		//Wait for Delay, copy Data and then next step
		IF NOT fbMBRead_FC4.bBusy AND NOT fbMBRead_FC4.bError AND timDelay.Q THEN
			//Connecotor State
			arrConnectorState[wConnectorInProgress] := arrBuffer_FC4[1];
			//Connector Power
			fbConvertWordToDord(wInputValue_1:= arrBuffer_FC4[5], wInputValue_2:= arrBuffer_FC4[6], eByteOrderForConvert:= eByteOrder.eBigEndian, dwOutputValue=> );
				arrPowerConnector[wConnectorInProgress] := fbConvertWordToDord.dwOutputValue;
			//Charging Time in Seconds
			arrChargingTime[wConnectorInProgress] := arrBuffer_FC4[7];
			//Energy Session
			arrEnergySession[wConnectorInProgress] := WORD_TO_REAL(arrBuffer_FC4[8]) / 100;
			//SOC from the Car
			arrSOCCar[wConnectorInProgress] := arrBuffer_FC4[9] / 100;
			//Go to Next Step
			fbMBRead_FC4.bExecute := FALSE;
				timDelay.IN := FALSE;		
					iStateModbusRead := 3;
		END_IF	

		//Error or Timeout
		IF FPError_FC_4.Q OR timTimeout.Q THEN
			iStateModbusError := 300;
		END_IF
		
	3://Wait 1 Step to reset the delay counter befor start to write
		iStateModbus_CP := iStateModbusRead;
		
			iStateModbusWrite := 1;
				//-1 because 0 is the Init Step for Read
				iStateModbusRead := - 1;
				
			//Error on Master, changes on Inputs or Timeout
		 	IF timTimeout.Q THEN 
				iStateModbusError := 300; 
					 
			END_IF
	
END_CASE

(*------------------------------------------------------------------Error and Warning----------------------------------------------------------------------------*)	
 
IF wStationState = 10 OR arrConnectorState[1] = 10 OR arrConnectorState[2] = 10 OR arrConnectorState[3] = 10 OR arrConnectorState[4] = 10 THEN bErrorCS := TRUE; ELSE bErrorCS := FALSE; END_IF  

IF timDissableFunctions.Q THEN fbCS.bWarning := TRUE; fbCS.iWarningCode := 0; ELSE fbCS.bWarning := FALSE; END_IF   
	IF Lynus_Standards.GVL_Energy.stNumberOfDevices.diNumberOfECS > Constants_Energy.diMaxNumberOfElectricChargingStations OR bErrorCS OR bMBTCPError THEN 
		fbCS.bError := TRUE;
	ELSE 
		fbCS.bError := FALSE;
			fbCS.iErrorCode := 0;
	END_IF

IF Lynus_Standards.GVL_Energy.stNumberOfDevices.diNumberOfECS > Constants_Energy.diMaxNumberOfElectricChargingStations THEN fbCS.iErrorCode := 1;
ELSIF bErrorCS OR bMBTCPError THEN fbCS.iErrorCode := 0; END_IF

(*------------------------------------------------------------------Logic----------------------------------------------------------------------------*)

//Calcualte the total SOC if we have more then 1 battery in our system
diNumberOfActiveBatterys := 0;
	dwSumSOC := 0;
		FOR liLPBatteryData := 1 TO Constants_Energy.diMaxNumberOfBatterys BY 1 DO
			IF Lynus_Standards.GVL_Energy.stDataOfBatterys[diNrOfEMS_IN,liLPBatteryData].bEnabled THEN diNumberOfActiveBatterys := diNumberOfActiveBatterys + 1; END_IF
				dwSumSOC := dwSumSOC + Lynus_Standards.GVL_Energy.stDataOfBatterys[diNrOfEMS_IN,liLPBatteryData].dwSOC;
		END_FOR
	
IF diNumberOfActiveBatterys > 0 THEN
	fbCS.dwBatterySOC := DINT_TO_DWORD(DWORD_TO_DINT(dwSumSOC) / diNumberOfActiveBatterys);
ELSE
	fbCS.dwBatterySOC := 100;	//When we have no battery in the ems system
END_IF

//Check if one or more Batterysystems or batteryinverter make island mode
diNumberOfBatteryInverterInEPO := 0;
	FOR liLPInEPO := 1 TO Constants_Energy.diMaxNumberOfBatteryInverters BY 1 DO
		IF Lynus_Standards.GVL_Energy.stDataOfBatteryInverters[diNrOfEMS_IN,liLPInEPO].bWorkOnIslandMode THEN fbCS.bEPOIsActive := TRUE; diNumberOfBatteryInverterInEPO := diNumberOfBatteryInverterInEPO + 1; END_IF
	END_FOR 
		IF diNumberOfBatteryInverterInEPO <= 0 THEN fbCS.bEPOIsActive := FALSE; END_IF

//Digital input for external lock signal
fbDIExternalLock(bInvers:= FALSE, bSignal=> );

//Car connected to the ECS  
IF arrConnectorState[1] = 2 OR arrConnectorState[2] = 2 OR arrConnectorState[3] = 2 OR arrConnectorState[4] = 2 OR
	 arrConnectorState[1] = 3 OR arrConnectorState[2] = 3 OR arrConnectorState[3] = 3 OR arrConnectorState[4] = 3 OR 
		arrConnectorState[1] = 6 OR arrConnectorState[2] = 6 OR arrConnectorState[3] = 6 OR arrConnectorState[4] = 6 THEN 
		fbCS.bCarConnected := TRUE; 
ELSE 
		fbCS.bCarConnected := FALSE; 
END_IF 

//Charging time and SOC from the Car
fbCS.arrSocketChargingTimeInput[1] :=  arrChargingTime[1] / 60;
fbCS.arrSocketChargingTimeInput[2] :=  arrChargingTime[2] / 60;
fbCS.arrSocketChargingTimeInput[3] :=  arrChargingTime[3] / 60;
fbCS.arrSocketChargingTimeInput[4] :=  arrChargingTime[4] / 60;

fbCS.arrSOCCar[1] := arrSOCCar[1];
fbCS.arrSOCCar[2] := arrSOCCar[2];
fbCS.arrSOCCar[3] := arrSOCCar[3];
fbCS.arrSOCCar[4] := arrSOCCar[4];

//Mode 3 State
fbCS.arrSocketMode3StateECS[1] := '';
fbCS.arrSocketMode3StateECS[2] := '';
fbCS.arrSocketMode3StateECS[3] := '';
fbCS.arrSocketMode3StateECS[4] := '';
//ECS is Free
IF arrConnectorState[1] = 0 THEN fbCS.arrSocketMode3StateECS[1] := 'A'; END_IF
IF arrConnectorState[2] = 0 THEN fbCS.arrSocketMode3StateECS[2] := 'A'; END_IF
IF arrConnectorState[3] = 0 THEN fbCS.arrSocketMode3StateECS[3] := 'A'; END_IF
IF arrConnectorState[4] = 0 THEN fbCS.arrSocketMode3StateECS[4] := 'A'; END_IF
//ECS Car Connected
IF arrConnectorState[1] = 2 OR arrConnectorState[1] = 6 THEN fbCS.arrSocketMode3StateECS[1] := 'B1'; END_IF
IF arrConnectorState[2] = 2 OR arrConnectorState[2] = 6 THEN fbCS.arrSocketMode3StateECS[2] := 'B1'; END_IF
IF arrConnectorState[3] = 2 OR arrConnectorState[3] = 6 THEN fbCS.arrSocketMode3StateECS[3] := 'B1'; END_IF
IF arrConnectorState[4] = 2 OR arrConnectorState[4] = 6 THEN fbCS.arrSocketMode3StateECS[4] := 'B1'; END_IF
//ECS Car is Charging
IF arrConnectorState[1] = 3 THEN fbCS.arrSocketMode3StateECS[1] := 'C2'; END_IF
IF arrConnectorState[2] = 3 THEN fbCS.arrSocketMode3StateECS[2] := 'C2'; END_IF
IF arrConnectorState[3] = 3 THEN fbCS.arrSocketMode3StateECS[3] := 'C2'; END_IF
IF arrConnectorState[4] = 3 THEN fbCS.arrSocketMode3StateECS[4] := 'C2'; END_IF

//Functionblock ECS
fbCS(
	bEnable:= bEnable AND NOT timDissableFunctions.Q, 
	bError:= ,
	bWarning := ,
	bEPOIsActive:= , 
	bExternalLock:= fbDIExternalLock.bSignal, 
	bCarConnected:= , 
	bWriteWithDelay:= TRUE, 
	bCalculateEnergySession:= ,
	iErrorCode:= , 
	iWarningCode:= , 
	arrSocketChargingTimeInput:= ,
	arrSOCCar:= , 
	dwBatterySOC:= , 
	lrTotalCounterEnergy_Consumption:= , 
	lrTotalCounterEnergy_Production:= , 
	lrCounterEnergyT1_Consumption:= , 
	lrCounterEnergyT2_Consumption:= , 
	lrCounterEnergyT1_Production:= , 
	lrCounterEnergyT2_Production:= , 
	lrTotalPowerECS:= , 
	arrSocketEnergySession:= ,
	rTargetPower:= Lynus_Standards.GVL_Energy.stDataElectricChargingStations[diNrOfEMS_IN,diNrOfECS_OUT].rTargetPowerEMS, 
	rSupplyVoltage:= 692, 
	rMinCurrent:= 7.5, 
	tTimDelayOutput:= T#5S, 
	tDelayError:= T#5S,
	arrSocketMode3StateECS:= ,
	arrSocketPowerECS:= ,
	stSetupECS:= stSetupECS, 
	stDataECSOut=> , 
	stDataECSOutDelay=> stDataECS);

dwTargetPower := REAL_TO_DWORD((stSetupECS.rMaxPower * fbCS.stDataECSOut.rTargetPower) / 100);
	dwTargetPower := dwTargetPower * 1000;

//Real time Power for Output
lrTotalPowerECSRealTime := fbCS.stDataECSOut.lrTotalPower;
	
(*------------------------------------------------------------------------------------------State Machine Write---------------------------------------------------------------------------------------------*)	

CASE iStateModbusWrite OF	

	1://Set the charging power (Reg 0)
		iStateModbus_CP := iStateModbusWrite;
		
			fbMBWrite_FC16.nQuantity := 2;
				fbMBWrite_FC16.nMBAddr := 0;
					fbMBWrite_FC16.bExecute := TRUE;
						fbMBWrite_FC16.nUnitID := byUnitID;
		
		//Prepear the sending Data. Charging Power for the charging station. 
		//Charging power
		fbConvertDwordToWord(dwInputValue:= dwTargetPower, eByteOrderForConvert:= eByteOrder.eBigEndian, wOutputValue_1=> arrBuffer_FC16[1], wOutputValue_2=> arrBuffer_FC16[2]);
		
		IF fbMBWrite_FC16.bBusy THEN timDelay.IN := TRUE; END_IF

		//Wait for Delay and then next step
		IF NOT fbMBWrite_FC16.bBusy AND NOT fbMBWrite_FC16.bError AND timDelay.Q THEN
			fbMBWrite_FC16.bExecute := FALSE;
				timDelay.IN := FALSE;
					bMBTCPError := FALSE; 
						//Restart from new with the Read out part
						iStateModbusRead := 1;
							iStateModbusWrite := 0;
								wConnectorInProgress := wConnectorInProgress + 1;
									IF wConnectorInProgress > 4 OR wConnectorInProgress > wNumberOfConnectors THEN wConnectorInProgress := 1; END_IF
		END_IF
				
		//Error or Timout
		IF FPError_FC_16.Q OR timTimeout.Q THEN
			iStateModbusError := 300;
		END_IF
		
END_CASE	
	
(*------------------------------------------------------------------------------------------State Machine Error---------------------------------------------------------------------------------------------*)	

CASE iStateModbusError OF
	
	300://Error
		iStateModbus_CP := iStateModbusError;
			timDelay.IN := FALSE;
				fbMBRead_FC4.bExecute := FALSE;
					fbMBWrite_FC16.bExecute := FALSE;
						bMBTCPError := TRUE; 		
							//Restart from new with the Read out part after an Error
							iStateModbusRead := 1;	
								iStateModbusError := 0;
									iStateModbusWrite := 0;
						
END_CASE

(*------------------------------------------------------------------------------------------Modbus TCP Functions---------------------------------------------------------------------------------------------*)

fbMBRead_FC4(sIPAddr:= sIPAdress, nTCPPort:= 502,cbLength:= SIZEOF(arrBuffer_FC4), pDestAddr:= ADR(arrBuffer_FC4), tTimeout:= T#10S );
	FPError_FC_4(CLK:= fbMBRead_FC4.bError, Q=> );		

fbMBWrite_FC16(sIPAddr:= sIPAdress, nTCPPort:= 502, cbLength:= SIZEOF(arrBuffer_FC16), pSrcAddr:= ADR(arrBuffer_FC16), tTimeout:= T#10S);	
	FPError_FC_16(CLK:= fbMBWrite_FC16.bError, Q=> );

(*-----------------------------------------------------------Handle data to Global structure for electric charging stations-----------------------------------------------------------------*)

//Delte al old Data on GVL after a online change or change on the variable diNrOfEMS_IDOD
IF diNrOfEMS_IN <> diNrOfEMS_IN_CP AND iStateGVLData = 0 THEN iStateGVLData := 10; END_IF 

CASE iStateGVLData OF
	
	0://Init Step
		byWaitInStep := 0;
			diCounterForGVL := 1;
	
	1://Wait for 4 Steps before clean al Data on GVL
		byWaitInStep := byWaitInStep + 1;
			IF byWaitInStep >= 4 AND fbNumberDevice.bNumberIsCalculatet THEN iStateGVLData := 2; END_IF
				//To much Devices, back to the Init step
				IF byWaitInStep >= 4 AND NOT fbNumberDevice.bNumberIsCalculatet THEN iStateGVLData := 0; END_IF	
			
	2://Clear all Data in GVL
		FOR diLPForGVL := 1 TO Constants_Energy.diMaxNumberOfEMS BY 1 DO 
			Lynus_Standards.GVL_Energy.stDataElectricChargingStations[diLPForGVL,diCounterForGVL].bEnabled := FALSE;
				Lynus_Standards.GVL_Energy.stDataElectricChargingStations[diLPForGVL,diCounterForGVL].bIsControllable := FALSE;
					Lynus_Standards.GVL_Energy.stDataElectricChargingStations[diLPForGVL,diCounterForGVL].byErrorWarning := 0;
						Lynus_Standards.GVL_Energy.stDataElectricChargingStations[diLPForGVL,diCounterForGVL].byPriority := 0;
							Lynus_Standards.GVL_Energy.stDataElectricChargingStations[diLPForGVL,diCounterForGVL].lrPower := 0;
								Lynus_Standards.GVL_Energy.stDataElectricChargingStations[diLPForGVL,diCounterForGVL].lrPowerConsumption := 0;
									Lynus_Standards.GVL_Energy.stDataElectricChargingStations[diLPForGVL,diCounterForGVL].lrPowerProduction := 0;
										Lynus_Standards.GVL_Energy.stDataElectricChargingStations[diLPForGVL,diCounterForGVL].rMaxPower := 0;
											//Set also the target value from ems back here to 0 and not in EMS function because EMS is in Standy when we have a online change (Problem when we delete a ems function and make a online change)
											Lynus_Standards.GVL_Energy.stDataElectricChargingStations[diLPForGVL,diCounterForGVL].rTargetPowerEMS := 0;	
		END_FOR
		
			//Counter for ECS
			diCounterForGVL := diCounterForGVL + 1;
				diCounterForGVL := LIMIT(0,diCounterForGVL,Constants_Energy.diMaxNumberOfElectricChargingStations);
					//Back to the init step
					IF diCounterForGVL >= Constants_Energy.diMaxNumberOfElectricChargingStations THEN iStateGVLData := 0; END_IF

	10://Clear old Data on GVL 		
		Lynus_Standards.GVL_Energy.stDataElectricChargingStations[diNrOfEMS_IN_CP,diNrOfECS_OUT].bEnabled := FALSE;
			Lynus_Standards.GVL_Energy.stDataElectricChargingStations[diNrOfEMS_IN_CP,diNrOfECS_OUT].bIsControllable := FALSE;
				Lynus_Standards.GVL_Energy.stDataElectricChargingStations[diNrOfEMS_IN_CP,diNrOfECS_OUT].byErrorWarning := 0;
					Lynus_Standards.GVL_Energy.stDataElectricChargingStations[diNrOfEMS_IN_CP,diNrOfECS_OUT].byPriority := 0;
						Lynus_Standards.GVL_Energy.stDataElectricChargingStations[diNrOfEMS_IN_CP,diNrOfECS_OUT].lrPower := 0;
							Lynus_Standards.GVL_Energy.stDataElectricChargingStations[diNrOfEMS_IN_CP,diNrOfECS_OUT].lrPowerConsumption := 0;
								Lynus_Standards.GVL_Energy.stDataElectricChargingStations[diNrOfEMS_IN_CP,diNrOfECS_OUT].lrPowerProduction := 0;
									Lynus_Standards.GVL_Energy.stDataElectricChargingStations[diNrOfEMS_IN_CP,diNrOfECS_OUT].rMaxPower := 0;
									
		diNrOfEMS_IN_CP := diNrOfEMS_IN;
			//Back to the init step
			iStateGVLData := 0;

END_CASE 	 

IF diNrOfECS_OUT > 0 AND fbNumberDevice.bNumberIsCalculatet AND diNrOfEMS_IN > 0 THEN
	Lynus_Standards.GVL_Energy.stDataElectricChargingStations[diNrOfEMS_IN,diNrOfECS_OUT].bEnabled := fbCS.stDataECSOut.bEnabled;
		Lynus_Standards.GVL_Energy.stDataElectricChargingStations[diNrOfEMS_IN,diNrOfECS_OUT].bIsControllable := TRUE;
			Lynus_Standards.GVL_Energy.stDataElectricChargingStations[diNrOfEMS_IN,diNrOfECS_OUT].byErrorWarning := fbCS.stDataECSOut.byErrorWarning;
				Lynus_Standards.GVL_Energy.stDataElectricChargingStations[diNrOfEMS_IN,diNrOfECS_OUT].byPriority := fbCS.stDataECSOut.byPriority;
					Lynus_Standards.GVL_Energy.stDataElectricChargingStations[diNrOfEMS_IN,diNrOfECS_OUT].lrPower := fbCS.stDataECSOut.lrTotalPower;
						Lynus_Standards.GVL_Energy.stDataElectricChargingStations[diNrOfEMS_IN,diNrOfECS_OUT].lrPowerConsumption := fbCS.stDataECSOut.lrTotalPowerConsumption;
							Lynus_Standards.GVL_Energy.stDataElectricChargingStations[diNrOfEMS_IN,diNrOfECS_OUT].lrPowerProduction := fbCS.stDataECSOut.lrTotalPowerProduction;
								Lynus_Standards.GVL_Energy.stDataElectricChargingStations[diNrOfEMS_IN,diNrOfECS_OUT].rMaxPower := fbCS.stDataECSOut.rMaxPower;	
END_IF 

(*----------------------------------------------------------Save persistent data----------------------------------------------------------------*)

arrPD[1](lrValue:= BOOL_TO_LREAL(bEnable), bEventBasedActive=> );
arrPD[2](lrValue:= BOOL_TO_LREAL(bPowerDataInvers), bEventBasedActive=> );
arrPD[3](lrValue:= DINT_TO_LREAL(diNrOfEMS_IN), bEventBasedActive=> );
arrPD[4](lrValue:= DINT_TO_LREAL(diNrOfEM_IN_CS), bEventBasedActive=> );
arrPD[5](lrValue:= BOOL_TO_LREAL(stSetupECS.bManualyOn), bEventBasedActive=> );
arrPD[6](lrValue:= BOOL_TO_LREAL(stSetupECS.bOnEmergPowerOff), bEventBasedActive=> );
arrPD[7](lrValue:= BYTE_TO_LREAL(stSetupECS.byCSMinPower), bEventBasedActive=> );
arrPD[8](lrValue:= BYTE_TO_LREAL(stSetupECS.byDisableSOC), bEventBasedActive=> );
arrPD[9](lrValue:= BYTE_TO_LREAL(stSetupECS.byEnableSOC), bEventBasedActive=> );
arrPD[10](lrValue:= BYTE_TO_LREAL(stSetupECS.byManualyTargetPower), bEventBasedActive=> );
arrPD[11](lrValue:= BYTE_TO_LREAL(stSetupECS.byPriority), bEventBasedActive=> );
arrPD[12](lrValue:= REAL_TO_LREAL(stSetupECS.rMaxPower), bEventBasedActive=> );
arrPD[13](lrValue:= DINT_TO_LREAL(diNrOfEMS_IN_CP), bEventBasedActive=> );
arrPD[14](lrValue:= BYTE_TO_LREAL(byUnitID), bEventBasedActive=> );
fbPDString(sText:= sIPAdress, bEventBasedActive=> );

END_FUNCTION_BLOCK

// ---- POUs/prgCS2.TcPOU
PROGRAM prgCS2
VAR
	fbAlfen1					: FB_ECS_Alfen_NG9xx_Platform;						//{#lynus.ag#()}
	fbAlfen2					: FB_ECS_Alfen_NG9xx_Platform;						//{#lynus.ag#()}
	fbAlfen3					: FB_ECS_Alfen_NG9xx_Platform;						//{#lynus.ag#()}
	fbAlfen4					: FB_ECS_Alfen_NG9xx_Platform;						//{#lynus.ag#()}
	fbAlfen5					: FB_ECS_Alfen_NG9xx_Platform;						//{#lynus.ag#()}
	fbAlfen6					: FB_ECS_Alfen_NG9xx_Platform;						//{#lynus.ag#()}
	fbAlfen7					: FB_ECS_Alfen_NG9xx_Platform;						//{#lynus.ag#()}
	fbAlfen8					: FB_ECS_Alfen_NG9xx_Platform;						//{#lynus.ag#()}
	fbAlfen9					: FB_ECS_Alfen_NG9xx_Platform;						//{#lynus.ag#()}
	fbAlfen10					: FB_ECS_Alfen_NG9xx_Platform;						//{#lynus.ag#()}
	
	bSManualyOn_UV1_1			: BOOL;												//{#lynus.ag#()}
	bySManualyTargetPowerUV1_1	: BYTE;												//{#lynus.ag#()}
	byErrorWarningUV1_1			: BYTE;												//{#lynus.ag#()}
	rChargingTimeInMinUV1_1		: REAL;												//{#lynus.ag#()}
	lrPowerUV1_1				: LREAL;											//{#lynus.ag#()}
	wStateUV1_1					: WORD;												//{#lynus.ag#()}
	lrEnergySessionUV1_1		: LREAL;											//{#lynus.ag#()}
	lrTotalEnergyUV1_1			: LREAL;											//{#lynus.ag#()}
	
	bSManualyOn_UV1_2			: BOOL;												//{#lynus.ag#()}
	bySManualyTargetPowerUV1_2	: BYTE;												//{#lynus.ag#()}
	byErrorWarningUV1_2			: BYTE;												//{#lynus.ag#()}
	rChargingTimeInMinUV1_2		: REAL;												//{#lynus.ag#()}
	lrPowerUV1_2				: LREAL;											//{#lynus.ag#()}
	wStateUV1_2					: WORD;												//{#lynus.ag#()}
	lrEnergySessionUV1_2		: LREAL;											//{#lynus.ag#()}
	lrTotalEnergyUV1_2			: LREAL;											//{#lynus.ag#()}
	
	bSManualyOn_UV1_3			: BOOL;												//{#lynus.ag#()}
	bySManualyTargetPowerUV1_3	: BYTE;												//{#lynus.ag#()}
	byErrorWarningUV1_3			: BYTE;												//{#lynus.ag#()}
	rChargingTimeInMinUV1_3		: REAL;												//{#lynus.ag#()}
	lrPowerUV1_3				: LREAL;											//{#lynus.ag#()}
	wStateUV1_3					: WORD;												//{#lynus.ag#()}
	lrEnergySessionUV1_3		: LREAL;											//{#lynus.ag#()}
	lrTotalEnergyUV1_3			: LREAL;											//{#lynus.ag#()}
	
	bSManualyOn_UV1_4			: BOOL;												//{#lynus.ag#()}
	bySManualyTargetPowerUV1_4	: BYTE;												//{#lynus.ag#()}
	byErrorWarningUV1_4			: BYTE;												//{#lynus.ag#()}
	rChargingTimeInMinUV1_4		: REAL;												//{#lynus.ag#()}
	lrPowerUV1_4				: LREAL;											//{#lynus.ag#()}
	wStateUV1_4					: WORD;												//{#lynus.ag#()}
	lrEnergySessionUV1_4		: LREAL;											//{#lynus.ag#()}
	lrTotalEnergyUV1_4			: LREAL;											//{#lynus.ag#()}
	
	bSManualyOn_UV1_5			: BOOL;												//{#lynus.ag#()}
	bySManualyTargetPowerUV1_5	: BYTE;												//{#lynus.ag#()}
	byErrorWarningUV1_5			: BYTE;												//{#lynus.ag#()}
	rChargingTimeInMinUV1_5		: REAL;												//{#lynus.ag#()}
	lrPowerUV1_5				: LREAL;											//{#lynus.ag#()}
	wStateUV1_5					: WORD;												//{#lynus.ag#()}
	lrEnergySessionUV1_5		: LREAL;											//{#lynus.ag#()}
	lrTotalEnergyUV1_5			: LREAL;											//{#lynus.ag#()}
	
	bSManualyOn_UV1_6			: BOOL;												//{#lynus.ag#()}
	bySManualyTargetPowerUV1_6	: BYTE;												//{#lynus.ag#()}
	byErrorWarningUV1_6			: BYTE;												//{#lynus.ag#()}
	rChargingTimeInMinUV1_6		: REAL;												//{#lynus.ag#()}
	lrPowerUV1_6				: LREAL;											//{#lynus.ag#()}
	wStateUV1_6					: WORD;												//{#lynus.ag#()}
	lrEnergySessionUV1_6		: LREAL;											//{#lynus.ag#()}
	lrTotalEnergyUV1_6			: LREAL;											//{#lynus.ag#()}
	
	bSManualyOn_UV1_7			: BOOL;												//{#lynus.ag#()}
	bySManualyTargetPowerUV1_7	: BYTE;												//{#lynus.ag#()}
	byErrorWarningUV1_7			: BYTE;												//{#lynus.ag#()}
	rChargingTimeInMinUV1_7		: REAL;												//{#lynus.ag#()}
	lrPowerUV1_7				: LREAL;											//{#lynus.ag#()}
	wStateUV1_7					: WORD;												//{#lynus.ag#()}
	lrEnergySessionUV1_7		: LREAL;											//{#lynus.ag#()}
	lrTotalEnergyUV1_7			: LREAL;											//{#lynus.ag#()}
	
	bSManualyOn_UV1_8			: BOOL;												//{#lynus.ag#()}
	bySManualyTargetPowerUV1_8	: BYTE;												//{#lynus.ag#()}
	byErrorWarningUV1_8			: BYTE;												//{#lynus.ag#()}
	rChargingTimeInMinUV1_8		: REAL;												//{#lynus.ag#()}
	lrPowerUV1_8				: LREAL;											//{#lynus.ag#()}
	wStateUV1_8					: WORD;												//{#lynus.ag#()}
	lrEnergySessionUV1_8		: LREAL;											//{#lynus.ag#()}
	lrTotalEnergyUV1_8			: LREAL;											//{#lynus.ag#()}
	
	bSManualyOn_UV1_9			: BOOL;												//{#lynus.ag#()}
	bySManualyTargetPowerUV1_9	: BYTE;												//{#lynus.ag#()}
	byErrorWarningUV1_9			: BYTE;												//{#lynus.ag#()}
	rChargingTimeInMinUV1_9		: REAL;												//{#lynus.ag#()}
	lrPowerUV1_9				: LREAL;											//{#lynus.ag#()}
	wStateUV1_9					: WORD;												//{#lynus.ag#()}
	lrEnergySessionUV1_9		: LREAL;											//{#lynus.ag#()}
	lrTotalEnergyUV1_9			: LREAL;											//{#lynus.ag#()}
	
	bSManualyOn_UV1_10			: BOOL;												//{#lynus.ag#()}
	bySManualyTargetPowerUV1_10	: BYTE;												//{#lynus.ag#()}
	byErrorWarningUV1_10		: BYTE;												//{#lynus.ag#()}
	rChargingTimeInMinUV1_10	: REAL;												//{#lynus.ag#()}
	lrPowerUV1_10				: LREAL;											//{#lynus.ag#()}
	wStateUV1_10				: WORD;												//{#lynus.ag#()}
	lrEnergySessionUV1_10		: LREAL;											//{#lynus.ag#()}
	lrTotalEnergyUV1_10			: LREAL;											//{#lynus.ag#()}
END_VAR
VAR PERSISTENT
	bManualyOnUV1_1				: BOOL;												//{#lynus.ag#()}
	byManualyTargetPowerUV1_1	: BYTE;												//{#lynus.ag#()}
	
	bManualyOnUV1_2				: BOOL;												//{#lynus.ag#()}
	byManualyTargetPowerUV1_2	: BYTE;												//{#lynus.ag#()}
	
	bManualyOnUV1_3				: BOOL;												//{#lynus.ag#()}
	byManualyTargetPowerUV1_3	: BYTE;												//{#lynus.ag#()}
	
	bManualyOnUV1_4				: BOOL;												//{#lynus.ag#()}
	byManualyTargetPowerUV1_4	: BYTE;												//{#lynus.ag#()}
	
	bManualyOnUV1_5				: BOOL;												//{#lynus.ag#()}
	byManualyTargetPowerUV1_5	: BYTE;												//{#lynus.ag#()}
	
	bManualyOnUV1_6				: BOOL;												//{#lynus.ag#()}
	byManualyTargetPowerUV1_6	: BYTE;												//{#lynus.ag#()}
	
	bManualyOnUV1_7				: BOOL;												//{#lynus.ag#()}
	byManualyTargetPowerUV1_7	: BYTE;												//{#lynus.ag#()}
	
	bManualyOnUV1_8				: BOOL;												//{#lynus.ag#()}
	byManualyTargetPowerUV1_8	: BYTE;												//{#lynus.ag#()}
	
	bManualyOnUV1_9				: BOOL;												//{#lynus.ag#()}
	byManualyTargetPowerUV1_9	: BYTE;												//{#lynus.ag#()}
	
	bManualyOnUV1_10			: BOOL;												//{#lynus.ag#()}
	byManualyTargetPowerUV1_10	: BYTE;												//{#lynus.ag#()}
END_VAR

(*---------------------------------------------CS1-----------------------------------------------------------*)

//Manual Power
fbAlfen1.stSetupECS.bManualyOn := bManualyOnUV1_1;
	fbAlfen1.stSetupECS.byManualyTargetPower := byManualyTargetPowerUV1_1;

fbAlfen1(
	bEnable:= , 
	bPowerDataInvers:= , 
	byElectricFuseLine:= , 
	byUnitID_Socket1:= 1, 
	byUnitID_Socket2:= , 
	byNumberOfSockets:= 1, 
	byNumberOfConnectionWire:= 1, 
	diNrOfEMS_IN:= prgEMS.fbEMS.diNrOfEMS_OUT, 
	diNrOfEM_IN_CS:= , 
	sIPAdress:= '192.168.1.125', 
	stSetupECS:= , 
	stDataECS=> , 
	diNrOfECS_OUT=> );

bSManualyOn_UV1_1 := fbAlfen1.stDataECS.bSManualyOn;
	bySManualyTargetPowerUV1_1 := fbAlfen1.stDataECS.bySManualyTargetPower;
		byErrorWarningUV1_1 := fbAlfen1.stDataECS.byErrorWarning;	
			rChargingTimeInMinUV1_1 := fbAlfen1.stDataECS.arrChargingTimeInMin[1];
				lrPowerUV1_1 := fbAlfen1.stDataECS.lrTotalPower;	
					wStateUV1_1 := fbAlfen1.stDataECS.arrSocketStateECS[1];
						lrEnergySessionUV1_1 := fbAlfen1.stDataECS.arrSocketEnergySession[1];
							lrTotalEnergyUV1_1 := fbAlfen1.stDataECS.lrTotalCounterEnergy_Consumption;	
	
(*---------------------------------------------CS2-----------------------------------------------------------*)
	
//Manual Power
fbAlfen2.stSetupECS.bManualyOn := bManualyOnUV1_2;
	fbAlfen2.stSetupECS.byManualyTargetPower := byManualyTargetPowerUV1_2;
	
fbAlfen2(
	bEnable:= , 
	bPowerDataInvers:= , 
	byElectricFuseLine:= , 
	byUnitID_Socket1:= 1, 
	byUnitID_Socket2:= , 
	byNumberOfSockets:= 1, 
	byNumberOfConnectionWire:= 1, 
	diNrOfEMS_IN:= prgEMS.fbEMS.diNrOfEMS_OUT, 
	diNrOfEM_IN_CS:= , 
	sIPAdress:= '192.168.1.195', 
	stSetupECS:= , 
	stDataECS=> , 
	diNrOfECS_OUT=> );

bSManualyOn_UV1_2 := fbAlfen2.stDataECS.bSManualyOn;
	bySManualyTargetPowerUV1_2 := fbAlfen2.stDataECS.bySManualyTargetPower;	
		byErrorWarningUV1_2 := fbAlfen2.stDataECS.byErrorWarning;
			rChargingTimeInMinUV1_2 := fbAlfen2.stDataECS.arrChargingTimeInMin[1];;
				lrPowerUV1_2 := fbAlfen2.stDataECS.lrTotalPower;	
					wStateUV1_2 := fbAlfen2.stDataECS.arrSocketStateECS[1];
						lrEnergySessionUV1_2 := fbAlfen2.stDataECS.arrSocketEnergySession[1];
							lrTotalEnergyUV1_2 := fbAlfen2.stDataECS.lrTotalCounterEnergy_Consumption;
	
(*---------------------------------------------CS3-----------------------------------------------------------*)	
	
//Manual Power
fbAlfen3.stSetupECS.bManualyOn := bManualyOnUV1_3;
	fbAlfen3.stSetupECS.byManualyTargetPower := byManualyTargetPowerUV1_3;
	
fbAlfen3(
	bEnable:= , 
	bPowerDataInvers:= , 
	byElectricFuseLine:= , 
	byUnitID_Socket1:= 1, 
	byUnitID_Socket2:= , 
	byNumberOfSockets:= 1, 
	byNumberOfConnectionWire:= 1, 
	diNrOfEMS_IN:= prgEMS.fbEMS.diNrOfEMS_OUT, 
	diNrOfEM_IN_CS:= , 
	sIPAdress:= '192.168.1.212',  
	stSetupECS:= , 
	stDataECS=> , 
	diNrOfECS_OUT=> );

bSManualyOn_UV1_3 := fbAlfen3.stDataECS.bSManualyOn;
	bySManualyTargetPowerUV1_3 := fbAlfen3.stDataECS.bySManualyTargetPower;
		byErrorWarningUV1_3 := fbAlfen3.stDataECS.byErrorWarning;
			rChargingTimeInMinUV1_3 := fbAlfen3.stDataECS.arrChargingTimeInMin[1];	
				lrPowerUV1_3 := fbAlfen3.stDataECS.lrTotalPower;	
					wStateUV1_3 := fbAlfen3.stDataECS.arrSocketStateECS[1];
						lrEnergySessionUV1_3 := fbAlfen3.stDataECS.arrSocketEnergySession[1];
							lrTotalEnergyUV1_3 := fbAlfen3.stDataECS.lrTotalCounterEnergy_Consumption;	
	
(*---------------------------------------------CS4-----------------------------------------------------------*)	
	
//Manual Power
fbAlfen4.stSetupECS.bManualyOn := bManualyOnUV1_4;
	fbAlfen4.stSetupECS.byManualyTargetPower := byManualyTargetPowerUV1_4;
	
fbAlfen4(
	bEnable:= , 
	bPowerDataInvers:= , 
	byElectricFuseLine:= , 
	byUnitID_Socket1:= 1, 
	byUnitID_Socket2:= , 
	byNumberOfSockets:= 1, 
	byNumberOfConnectionWire:= 1, 
	diNrOfEMS_IN:= prgEMS.fbEMS.diNrOfEMS_OUT, 
	diNrOfEM_IN_CS:= , 
	sIPAdress:= '192.168.1.140',  
	stSetupECS:= , 
	stDataECS=> , 
	diNrOfECS_OUT=> );

bSManualyOn_UV1_4 := fbAlfen4.stDataECS.bSManualyOn;
	bySManualyTargetPowerUV1_4 := fbAlfen4.stDataECS.bySManualyTargetPower;	
		byErrorWarningUV1_4 := fbAlfen4.stDataECS.byErrorWarning;
			rChargingTimeInMinUV1_4 := fbAlfen4.stDataECS.arrChargingTimeInMin[1];
				lrPowerUV1_4 := fbAlfen4.stDataECS.lrTotalPower;	
					wStateUV1_4 := fbAlfen4.stDataECS.arrSocketStateECS[1];
						lrEnergySessionUV1_4 := fbAlfen4.stDataECS.arrSocketEnergySession[1];
							lrTotalEnergyUV1_4 := fbAlfen4.stDataECS.lrTotalCounterEnergy_Consumption;
	
(*---------------------------------------------CS5-----------------------------------------------------------*)	
	
//Manual Power
fbAlfen5.stSetupECS.bManualyOn := bManualyOnUV1_5;
	fbAlfen5.stSetupECS.byManualyTargetPower := byManualyTargetPowerUV1_5;
	
fbAlfen5(
	bEnable:= , 
	bPowerDataInvers:= , 
	byElectricFuseLine:= , 
	byUnitID_Socket1:= 1, 
	byUnitID_Socket2:= , 
	byNumberOfSockets:= 1, 
	byNumberOfConnectionWire:= 1, 
	diNrOfEMS_IN:= prgEMS.fbEMS.diNrOfEMS_OUT, 
	diNrOfEM_IN_CS:= , 
	sIPAdress:= '192.168.1.222',  
	stSetupECS:= , 
	stDataECS=> , 
	diNrOfECS_OUT=> );

bSManualyOn_UV1_5 := fbAlfen5.stDataECS.bSManualyOn;
	bySManualyTargetPowerUV1_5 := fbAlfen5.stDataECS.bySManualyTargetPower;
		byErrorWarningUV1_5 := fbAlfen5.stDataECS.byErrorWarning;
			rChargingTimeInMinUV1_5 := fbAlfen5.stDataECS.arrChargingTimeInMin[1];
				lrPowerUV1_5 := fbAlfen5.stDataECS.lrTotalPower;	
					wStateUV1_5 := fbAlfen5.stDataECS.arrSocketStateECS[1];
						lrEnergySessionUV1_5 := fbAlfen5.stDataECS.arrSocketEnergySession[1];
							lrTotalEnergyUV1_5 := fbAlfen5.stDataECS.lrTotalCounterEnergy_Consumption;	
	
(*---------------------------------------------CS6-----------------------------------------------------------*)	
	
//Manual Power
fbAlfen6.stSetupECS.bManualyOn := bManualyOnUV1_6;
	fbAlfen6.stSetupECS.byManualyTargetPower := byManualyTargetPowerUV1_6;
	
fbAlfen6(
	bEnable:= , 
	bPowerDataInvers:= , 
	byElectricFuseLine:= , 
	byUnitID_Socket1:= 1, 
	byUnitID_Socket2:= , 
	byNumberOfSockets:= 1, 
	byNumberOfConnectionWire:= 1, 
	diNrOfEMS_IN:= prgEMS.fbEMS.diNrOfEMS_OUT, 
	diNrOfEM_IN_CS:= , 
	sIPAdress:= '192.168.1.196',  
	stSetupECS:= , 
	stDataECS=> , 
	diNrOfECS_OUT=> );

bSManualyOn_UV1_6 := fbAlfen6.stDataECS.bSManualyOn;
	bySManualyTargetPowerUV1_6 := fbAlfen6.stDataECS.bySManualyTargetPower;	
		byErrorWarningUV1_6 := fbAlfen6.stDataECS.byErrorWarning;
			rChargingTimeInMinUV1_6 := fbAlfen6.stDataECS.arrChargingTimeInMin[1];
				lrPowerUV1_6 := fbAlfen6.stDataECS.lrTotalPower;	
					wStateUV1_6 := fbAlfen6.stDataECS.arrSocketStateECS[1];
						lrEnergySessionUV1_6 := fbAlfen6.stDataECS.arrSocketEnergySession[1];
							lrTotalEnergyUV1_6 := fbAlfen6.stDataECS.lrTotalCounterEnergy_Consumption;
	
(*---------------------------------------------CS7-----------------------------------------------------------*)	
	
//Manual Power
fbAlfen7.stSetupECS.bManualyOn := bManualyOnUV1_7;
	fbAlfen7.stSetupECS.byManualyTargetPower := byManualyTargetPowerUV1_7;
	
fbAlfen7(
	bEnable:= , 
	bPowerDataInvers:= , 
	byElectricFuseLine:= , 
	byUnitID_Socket1:= 1, 
	byUnitID_Socket2:= , 
	byNumberOfSockets:= 1, 
	byNumberOfConnectionWire:= 1, 
	diNrOfEMS_IN:= prgEMS.fbEMS.diNrOfEMS_OUT, 
	diNrOfEM_IN_CS:= , 
	sIPAdress:= '192.168.1.127',  
	stSetupECS:= , 
	stDataECS=> , 
	diNrOfECS_OUT=> );

bSManualyOn_UV1_7 := fbAlfen7.stDataECS.bSManualyOn;
	bySManualyTargetPowerUV1_7 := fbAlfen7.stDataECS.bySManualyTargetPower;	
		byErrorWarningUV1_7 := fbAlfen7.stDataECS.byErrorWarning;
			rChargingTimeInMinUV1_7 := fbAlfen7.stDataECS.arrChargingTimeInMin[1];
				lrPowerUV1_7 := fbAlfen7.stDataECS.lrTotalPower;	
					wStateUV1_7 := fbAlfen7.stDataECS.arrSocketStateECS[1];
						lrEnergySessionUV1_7 := fbAlfen7.stDataECS.arrSocketEnergySession[1];
							lrTotalEnergyUV1_7 := fbAlfen7.stDataECS.lrTotalCounterEnergy_Consumption;
	
(*---------------------------------------------CS8-----------------------------------------------------------*)	
	
//Manual Power
fbAlfen8.stSetupECS.bManualyOn := bManualyOnUV1_8;
	fbAlfen8.stSetupECS.byManualyTargetPower := byManualyTargetPowerUV1_8;
	
fbAlfen8(
	bEnable:= , 
	bPowerDataInvers:= , 
	byElectricFuseLine:= , 
	byUnitID_Socket1:= 1, 
	byUnitID_Socket2:= , 
	byNumberOfSockets:= 1, 
	byNumberOfConnectionWire:= 1, 
	diNrOfEMS_IN:= prgEMS.fbEMS.diNrOfEMS_OUT, 
	diNrOfEM_IN_CS:= , 
	sIPAdress:= '192.168.1.237',  
	stSetupECS:= , 
	stDataECS=> , 
	diNrOfECS_OUT=> );

bSManualyOn_UV1_8 := fbAlfen8.stDataECS.bSManualyOn;
	bySManualyTargetPowerUV1_8 := fbAlfen8.stDataECS.bySManualyTargetPower;	
		byErrorWarningUV1_8 := fbAlfen8.stDataECS.byErrorWarning;
			rChargingTimeInMinUV1_8 := fbAlfen8.stDataECS.arrChargingTimeInMin[1];
				lrPowerUV1_8 := fbAlfen8.stDataECS.lrTotalPower;	
					wStateUV1_8 := fbAlfen8.stDataECS.arrSocketStateECS[1];
						lrEnergySessionUV1_8 := fbAlfen8.stDataECS.arrSocketEnergySession[1];
							lrTotalEnergyUV1_8 := fbAlfen8.stDataECS.lrTotalCounterEnergy_Consumption;
	
(*---------------------------------------------CS9-----------------------------------------------------------*)	
	
//Manual Power
fbAlfen9.stSetupECS.bManualyOn := bManualyOnUV1_9;
	fbAlfen9.stSetupECS.byManualyTargetPower := byManualyTargetPowerUV1_9;
	
fbAlfen9(
	bEnable:= , 
	bPowerDataInvers:= , 
	byElectricFuseLine:= , 
	byUnitID_Socket1:= 1, 
	byUnitID_Socket2:= , 
	byNumberOfSockets:= 1, 
	byNumberOfConnectionWire:= 1, 
	diNrOfEMS_IN:= prgEMS.fbEMS.diNrOfEMS_OUT, 
	diNrOfEM_IN_CS:= , 
	sIPAdress:= '192.168.1.112',  
	stSetupECS:= , 
	stDataECS=> , 
	diNrOfECS_OUT=> );

bSManualyOn_UV1_9 := fbAlfen9.stDataECS.bSManualyOn;
	bySManualyTargetPowerUV1_9 := fbAlfen9.stDataECS.bySManualyTargetPower;
		byErrorWarningUV1_9 := fbAlfen9.stDataECS.byErrorWarning;	
			rChargingTimeInMinUV1_9 := fbAlfen9.stDataECS.arrChargingTimeInMin[1];
				lrPowerUV1_9 := fbAlfen9.stDataECS.lrTotalPower;	
					wStateUV1_9 := fbAlfen9.stDataECS.arrSocketStateECS[1];
						lrEnergySessionUV1_9 := fbAlfen9.stDataECS.arrSocketEnergySession[1];
							lrTotalEnergyUV1_9 := fbAlfen9.stDataECS.lrTotalCounterEnergy_Consumption;
	
(*---------------------------------------------CS10-----------------------------------------------------------*)	
	
//Manual Power
fbAlfen10.stSetupECS.bManualyOn := bManualyOnUV1_10;
	fbAlfen10.stSetupECS.byManualyTargetPower := byManualyTargetPowerUV1_10;
	
fbAlfen10(
	bEnable:= , 
	bPowerDataInvers:= , 
	byElectricFuseLine:= , 
	byUnitID_Socket1:= 1, 
	byUnitID_Socket2:= , 
	byNumberOfSockets:= 1, 
	byNumberOfConnectionWire:= 1, 
	diNrOfEMS_IN:= prgEMS.fbEMS.diNrOfEMS_OUT, 
	diNrOfEM_IN_CS:= , 
	sIPAdress:= '192.168.1.203', 
	stSetupECS:= , 
	stDataECS=> , 
	diNrOfECS_OUT=> );

bSManualyOn_UV1_10 := fbAlfen10.stDataECS.bSManualyOn;
	bySManualyTargetPowerUV1_10 := fbAlfen10.stDataECS.bySManualyTargetPower;
		byErrorWarningUV1_10 := fbAlfen10.stDataECS.byErrorWarning;	
			rChargingTimeInMinUV1_10 := fbAlfen10.stDataECS.arrChargingTimeInMin[1];
				lrPowerUV1_10 := fbAlfen10.stDataECS.lrTotalPower;	
					wStateUV1_10 := fbAlfen10.stDataECS.arrSocketStateECS[1];
						lrEnergySessionUV1_10 := fbAlfen10.stDataECS.arrSocketEnergySession[1];
							lrTotalEnergyUV1_10 := fbAlfen10.stDataECS.lrTotalCounterEnergy_Consumption;

END_PROGRAM

// ---- POUs/prgCS3.TcPOU
PROGRAM prgCS3
VAR
	fbAlfen1					: FB_ECS_Alfen_NG9xx_Platform;						//{#lynus.ag#()}
	fbAlfen2					: FB_ECS_Alfen_NG9xx_Platform;						//{#lynus.ag#()}
	fbAlfen3					: FB_ECS_Alfen_NG9xx_Platform;						//{#lynus.ag#()}
	fbAlfen4					: FB_ECS_Alfen_NG9xx_Platform;						//{#lynus.ag#()}
	fbAlfen5					: FB_ECS_Alfen_NG9xx_Platform;						//{#lynus.ag#()}
	fbAlfen6					: FB_ECS_Alfen_NG9xx_Platform;						//{#lynus.ag#()}
	fbAlfen7					: FB_ECS_Alfen_NG9xx_Platform;						//{#lynus.ag#()}
	fbAlfen8					: FB_ECS_Alfen_NG9xx_Platform;						//{#lynus.ag#()}
	fbAlfen9					: FB_ECS_Alfen_NG9xx_Platform;						//{#lynus.ag#()}
	fbAlfen10					: FB_ECS_Alfen_NG9xx_Platform;						//{#lynus.ag#()}
	
	bSManualyOn_UV1_1			: BOOL;												//{#lynus.ag#()}
	bySManualyTargetPowerUV1_1	: BYTE;												//{#lynus.ag#()}
	byErrorWarningUV1_1			: BYTE;												//{#lynus.ag#()}
	rChargingTimeInMinUV1_1		: REAL;												//{#lynus.ag#()}
	lrPowerUV1_1				: LREAL;											//{#lynus.ag#()}
	wStateUV1_1					: WORD;												//{#lynus.ag#()}
	lrEnergySessionUV1_1		: LREAL;											//{#lynus.ag#()}
	lrTotalEnergyUV1_1			: LREAL;											//{#lynus.ag#()}
	
	bSManualyOn_UV1_2			: BOOL;												//{#lynus.ag#()}
	bySManualyTargetPowerUV1_2	: BYTE;												//{#lynus.ag#()}
	byErrorWarningUV1_2			: BYTE;												//{#lynus.ag#()}
	rChargingTimeInMinUV1_2		: REAL;												//{#lynus.ag#()}
	lrPowerUV1_2				: LREAL;											//{#lynus.ag#()}
	wStateUV1_2					: WORD;												//{#lynus.ag#()}
	lrEnergySessionUV1_2		: LREAL;											//{#lynus.ag#()}
	lrTotalEnergyUV1_2			: LREAL;											//{#lynus.ag#()}
	
	bSManualyOn_UV1_3			: BOOL;												//{#lynus.ag#()}
	bySManualyTargetPowerUV1_3	: BYTE;												//{#lynus.ag#()}
	byErrorWarningUV1_3			: BYTE;												//{#lynus.ag#()}
	rChargingTimeInMinUV1_3		: REAL;												//{#lynus.ag#()}
	lrPowerUV1_3				: LREAL;											//{#lynus.ag#()}
	wStateUV1_3					: WORD;												//{#lynus.ag#()}
	lrEnergySessionUV1_3		: LREAL;											//{#lynus.ag#()}
	lrTotalEnergyUV1_3			: LREAL;											//{#lynus.ag#()}
	
	bSManualyOn_UV1_4			: BOOL;												//{#lynus.ag#()}
	bySManualyTargetPowerUV1_4	: BYTE;												//{#lynus.ag#()}
	byErrorWarningUV1_4			: BYTE;												//{#lynus.ag#()}
	rChargingTimeInMinUV1_4		: REAL;												//{#lynus.ag#()}
	lrPowerUV1_4				: LREAL;											//{#lynus.ag#()}
	wStateUV1_4					: WORD;												//{#lynus.ag#()}
	lrEnergySessionUV1_4		: LREAL;											//{#lynus.ag#()}
	lrTotalEnergyUV1_4			: LREAL;											//{#lynus.ag#()}
	
	bSManualyOn_UV1_5			: BOOL;												//{#lynus.ag#()}
	bySManualyTargetPowerUV1_5	: BYTE;												//{#lynus.ag#()}
	byErrorWarningUV1_5			: BYTE;												//{#lynus.ag#()}
	rChargingTimeInMinUV1_5		: REAL;												//{#lynus.ag#()}
	lrPowerUV1_5				: LREAL;											//{#lynus.ag#()}
	wStateUV1_5					: WORD;												//{#lynus.ag#()}
	lrEnergySessionUV1_5		: LREAL;											//{#lynus.ag#()}
	lrTotalEnergyUV1_5			: LREAL;											//{#lynus.ag#()}
	
	bSManualyOn_UV1_6			: BOOL;												//{#lynus.ag#()}
	bySManualyTargetPowerUV1_6	: BYTE;												//{#lynus.ag#()}
	byErrorWarningUV1_6			: BYTE;												//{#lynus.ag#()}
	rChargingTimeInMinUV1_6		: REAL;												//{#lynus.ag#()}
	lrPowerUV1_6				: LREAL;											//{#lynus.ag#()}
	wStateUV1_6					: WORD;												//{#lynus.ag#()}
	lrEnergySessionUV1_6		: LREAL;											//{#lynus.ag#()}
	lrTotalEnergyUV1_6			: LREAL;											//{#lynus.ag#()}
	
	bSManualyOn_UV1_7			: BOOL;												//{#lynus.ag#()}
	bySManualyTargetPowerUV1_7	: BYTE;												//{#lynus.ag#()}
	byErrorWarningUV1_7			: BYTE;												//{#lynus.ag#()}
	rChargingTimeInMinUV1_7		: REAL;												//{#lynus.ag#()}
	lrPowerUV1_7				: LREAL;											//{#lynus.ag#()}
	wStateUV1_7					: WORD;												//{#lynus.ag#()}
	lrEnergySessionUV1_7		: LREAL;											//{#lynus.ag#()}
	lrTotalEnergyUV1_7			: LREAL;											//{#lynus.ag#()}
	
	bSManualyOn_UV1_8			: BOOL;												//{#lynus.ag#()}
	bySManualyTargetPowerUV1_8	: BYTE;												//{#lynus.ag#()}
	byErrorWarningUV1_8			: BYTE;												//{#lynus.ag#()}
	rChargingTimeInMinUV1_8		: REAL;												//{#lynus.ag#()}
	lrPowerUV1_8				: LREAL;											//{#lynus.ag#()}
	wStateUV1_8					: WORD;												//{#lynus.ag#()}
	lrEnergySessionUV1_8		: LREAL;											//{#lynus.ag#()}
	lrTotalEnergyUV1_8			: LREAL;											//{#lynus.ag#()}
	
	bSManualyOn_UV1_9			: BOOL;												//{#lynus.ag#()}
	bySManualyTargetPowerUV1_9	: BYTE;												//{#lynus.ag#()}
	byErrorWarningUV1_9			: BYTE;												//{#lynus.ag#()}
	rChargingTimeInMinUV1_9		: REAL;												//{#lynus.ag#()}
	lrPowerUV1_9				: LREAL;											//{#lynus.ag#()}
	wStateUV1_9					: WORD;												//{#lynus.ag#()}
	lrEnergySessionUV1_9		: LREAL;											//{#lynus.ag#()}
	lrTotalEnergyUV1_9			: LREAL;											//{#lynus.ag#()}
	
	bSManualyOn_UV1_10			: BOOL;												//{#lynus.ag#()}
	bySManualyTargetPowerUV1_10	: BYTE;												//{#lynus.ag#()}
	byErrorWarningUV1_10		: BYTE;												//{#lynus.ag#()}
	rChargingTimeInMinUV1_10	: REAL;												//{#lynus.ag#()}
	lrPowerUV1_10				: LREAL;											//{#lynus.ag#()}
	wStateUV1_10				: WORD;												//{#lynus.ag#()}
	lrEnergySessionUV1_10		: LREAL;											//{#lynus.ag#()}
	lrTotalEnergyUV1_10			: LREAL;											//{#lynus.ag#()}
END_VAR
VAR PERSISTENT
	bManualyOnUV1_1				: BOOL;												//{#lynus.ag#()}
	byManualyTargetPowerUV1_1	: BYTE;												//{#lynus.ag#()}
	
	bManualyOnUV1_2				: BOOL;												//{#lynus.ag#()}
	byManualyTargetPowerUV1_2	: BYTE;												//{#lynus.ag#()}
	
	bManualyOnUV1_3				: BOOL;												//{#lynus.ag#()}
	byManualyTargetPowerUV1_3	: BYTE;												//{#lynus.ag#()}
	
	bManualyOnUV1_4				: BOOL;												//{#lynus.ag#()}
	byManualyTargetPowerUV1_4	: BYTE;												//{#lynus.ag#()}
	
	bManualyOnUV1_5				: BOOL;												//{#lynus.ag#()}
	byManualyTargetPowerUV1_5	: BYTE;												//{#lynus.ag#()}
	
	bManualyOnUV1_6				: BOOL;												//{#lynus.ag#()}
	byManualyTargetPowerUV1_6	: BYTE;												//{#lynus.ag#()}
	
	bManualyOnUV1_7				: BOOL;												//{#lynus.ag#()}
	byManualyTargetPowerUV1_7	: BYTE;												//{#lynus.ag#()}
	
	bManualyOnUV1_8				: BOOL;												//{#lynus.ag#()}
	byManualyTargetPowerUV1_8	: BYTE;												//{#lynus.ag#()}
	
	bManualyOnUV1_9				: BOOL;												//{#lynus.ag#()}
	byManualyTargetPowerUV1_9	: BYTE;												//{#lynus.ag#()}
	
	bManualyOnUV1_10			: BOOL;												//{#lynus.ag#()}
	byManualyTargetPowerUV1_10	: BYTE;												//{#lynus.ag#()}
END_VAR

(*---------------------------------------------CS1-----------------------------------------------------------*)

//Manual Power
fbAlfen1.stSetupECS.bManualyOn := bManualyOnUV1_1;
	fbAlfen1.stSetupECS.byManualyTargetPower := byManualyTargetPowerUV1_1;

fbAlfen1(
	bEnable:= , 
	bPowerDataInvers:= , 
	byElectricFuseLine:= , 
	byUnitID_Socket1:= 1, 
	byUnitID_Socket2:= , 
	byNumberOfSockets:= 1, 
	byNumberOfConnectionWire:= 1, 
	diNrOfEMS_IN:= prgEMS.fbEMS.diNrOfEMS_OUT, 
	diNrOfEM_IN_CS:= , 
	sIPAdress:= '192.168.1.194', 
	stSetupECS:= , 
	stDataECS=> , 
	diNrOfECS_OUT=> );

bSManualyOn_UV1_1 := fbAlfen1.stDataECS.bSManualyOn;
	bySManualyTargetPowerUV1_1 := fbAlfen1.stDataECS.bySManualyTargetPower;
		byErrorWarningUV1_1 := fbAlfen1.stDataECS.byErrorWarning;	
			rChargingTimeInMinUV1_1 := fbAlfen1.stDataECS.arrChargingTimeInMin[1];
				lrPowerUV1_1 := fbAlfen1.stDataECS.lrTotalPower;	
					wStateUV1_1 := fbAlfen1.stDataECS.arrSocketStateECS[1];
						lrEnergySessionUV1_1 := fbAlfen1.stDataECS.arrSocketEnergySession[1];
							lrTotalEnergyUV1_1 := fbAlfen1.stDataECS.lrTotalCounterEnergy_Consumption;		
	
(*---------------------------------------------CS2-----------------------------------------------------------*)
	
//Manual Power
fbAlfen2.stSetupECS.bManualyOn := bManualyOnUV1_2;
	fbAlfen2.stSetupECS.byManualyTargetPower := byManualyTargetPowerUV1_2;
	
fbAlfen2(
	bEnable:= , 
	bPowerDataInvers:= , 
	byElectricFuseLine:= , 
	byUnitID_Socket1:= 1, 
	byUnitID_Socket2:= , 
	byNumberOfSockets:= 1, 
	byNumberOfConnectionWire:= 1, 
	diNrOfEMS_IN:= prgEMS.fbEMS.diNrOfEMS_OUT, 
	diNrOfEM_IN_CS:= , 
	sIPAdress:= '192.168.1.119', 
	stSetupECS:= , 
	stDataECS=> , 
	diNrOfECS_OUT=> );

bSManualyOn_UV1_2 := fbAlfen2.stDataECS.bSManualyOn;
	bySManualyTargetPowerUV1_2 := fbAlfen2.stDataECS.bySManualyTargetPower;	
		byErrorWarningUV1_2 := fbAlfen2.stDataECS.byErrorWarning;
			rChargingTimeInMinUV1_2 := fbAlfen2.stDataECS.arrChargingTimeInMin[1];;
				lrPowerUV1_2 := fbAlfen2.stDataECS.lrTotalPower;	
					wStateUV1_2 := fbAlfen2.stDataECS.arrSocketStateECS[1];
						lrEnergySessionUV1_2 := fbAlfen2.stDataECS.arrSocketEnergySession[1];
							lrTotalEnergyUV1_2 := fbAlfen2.stDataECS.lrTotalCounterEnergy_Consumption;
	
(*---------------------------------------------CS3-----------------------------------------------------------*)	
	
//Manual Power
fbAlfen3.stSetupECS.bManualyOn := bManualyOnUV1_3;
	fbAlfen3.stSetupECS.byManualyTargetPower := byManualyTargetPowerUV1_3;
	
fbAlfen3(
	bEnable:= , 
	bPowerDataInvers:= , 
	byElectricFuseLine:= , 
	byUnitID_Socket1:= 1, 
	byUnitID_Socket2:= , 
	byNumberOfSockets:= 1, 
	byNumberOfConnectionWire:= 1, 
	diNrOfEMS_IN:= prgEMS.fbEMS.diNrOfEMS_OUT, 
	diNrOfEM_IN_CS:= , 
	sIPAdress:= '192.168.1.217',  
	stSetupECS:= , 
	stDataECS=> , 
	diNrOfECS_OUT=> );

bSManualyOn_UV1_3 := fbAlfen3.stDataECS.bSManualyOn;
	bySManualyTargetPowerUV1_3 := fbAlfen3.stDataECS.bySManualyTargetPower;
		byErrorWarningUV1_3 := fbAlfen3.stDataECS.byErrorWarning;
			rChargingTimeInMinUV1_3 := fbAlfen3.stDataECS.arrChargingTimeInMin[1];	
				lrPowerUV1_3 := fbAlfen3.stDataECS.lrTotalPower;	
					wStateUV1_3 := fbAlfen3.stDataECS.arrSocketStateECS[1];
						lrEnergySessionUV1_3 := fbAlfen3.stDataECS.arrSocketEnergySession[1];
							lrTotalEnergyUV1_3 := fbAlfen3.stDataECS.lrTotalCounterEnergy_Consumption;	
	
(*---------------------------------------------CS4-----------------------------------------------------------*)	
	
//Manual Power
fbAlfen4.stSetupECS.bManualyOn := bManualyOnUV1_4;
	fbAlfen4.stSetupECS.byManualyTargetPower := byManualyTargetPowerUV1_4;
	
fbAlfen4(
	bEnable:= , 
	bPowerDataInvers:= , 
	byElectricFuseLine:= , 
	byUnitID_Socket1:= 1, 
	byUnitID_Socket2:= , 
	byNumberOfSockets:= 1, 
	byNumberOfConnectionWire:= 1, 
	diNrOfEMS_IN:= prgEMS.fbEMS.diNrOfEMS_OUT, 
	diNrOfEM_IN_CS:= , 
	sIPAdress:= '192.168.1.230',  
	stSetupECS:= , 
	stDataECS=> , 
	diNrOfECS_OUT=> );

bSManualyOn_UV1_4 := fbAlfen4.stDataECS.bSManualyOn;
	bySManualyTargetPowerUV1_4 := fbAlfen4.stDataECS.bySManualyTargetPower;	
		byErrorWarningUV1_4 := fbAlfen4.stDataECS.byErrorWarning;
			rChargingTimeInMinUV1_4 := fbAlfen4.stDataECS.arrChargingTimeInMin[1];
				lrPowerUV1_4 := fbAlfen4.stDataECS.lrTotalPower;	
					wStateUV1_4 := fbAlfen4.stDataECS.arrSocketStateECS[1];
						lrEnergySessionUV1_4 := fbAlfen4.stDataECS.arrSocketEnergySession[1];
							lrTotalEnergyUV1_4 := fbAlfen4.stDataECS.lrTotalCounterEnergy_Consumption;
	
(*---------------------------------------------CS5-----------------------------------------------------------*)	
	
//Manual Power
fbAlfen5.stSetupECS.bManualyOn := bManualyOnUV1_5;
	fbAlfen5.stSetupECS.byManualyTargetPower := byManualyTargetPowerUV1_5;
	
fbAlfen5(
	bEnable:= , 
	bPowerDataInvers:= , 
	byElectricFuseLine:= , 
	byUnitID_Socket1:= 1, 
	byUnitID_Socket2:= , 
	byNumberOfSockets:= 1, 
	byNumberOfConnectionWire:= 1, 
	diNrOfEMS_IN:= prgEMS.fbEMS.diNrOfEMS_OUT, 
	diNrOfEM_IN_CS:= , 
	sIPAdress:= '192.168.1.174',  
	stSetupECS:= , 
	stDataECS=> , 
	diNrOfECS_OUT=> );

bSManualyOn_UV1_5 := fbAlfen5.stDataECS.bSManualyOn;
	bySManualyTargetPowerUV1_5 := fbAlfen5.stDataECS.bySManualyTargetPower;
		byErrorWarningUV1_5 := fbAlfen5.stDataECS.byErrorWarning;
			rChargingTimeInMinUV1_5 := fbAlfen5.stDataECS.arrChargingTimeInMin[1];
				lrPowerUV1_5 := fbAlfen5.stDataECS.lrTotalPower;	
					wStateUV1_5 := fbAlfen5.stDataECS.arrSocketStateECS[1];
						lrEnergySessionUV1_5 := fbAlfen5.stDataECS.arrSocketEnergySession[1];
							lrTotalEnergyUV1_5 := fbAlfen5.stDataECS.lrTotalCounterEnergy_Consumption;	
	
(*---------------------------------------------CS6-----------------------------------------------------------*)	
	
//Manual Power
fbAlfen6.stSetupECS.bManualyOn := bManualyOnUV1_6;
	fbAlfen6.stSetupECS.byManualyTargetPower := byManualyTargetPowerUV1_6;
	
fbAlfen6(
	bEnable:= , 
	bPowerDataInvers:= , 
	byElectricFuseLine:= , 
	byUnitID_Socket1:= 1, 
	byUnitID_Socket2:= , 
	byNumberOfSockets:= 1, 
	byNumberOfConnectionWire:= 1, 
	diNrOfEMS_IN:= prgEMS.fbEMS.diNrOfEMS_OUT, 
	diNrOfEM_IN_CS:= , 
	sIPAdress:= '192.168.1.229',  
	stSetupECS:= , 
	stDataECS=> , 
	diNrOfECS_OUT=> );

bSManualyOn_UV1_6 := fbAlfen6.stDataECS.bSManualyOn;
	bySManualyTargetPowerUV1_6 := fbAlfen6.stDataECS.bySManualyTargetPower;	
		byErrorWarningUV1_6 := fbAlfen6.stDataECS.byErrorWarning;
			rChargingTimeInMinUV1_6 := fbAlfen6.stDataECS.arrChargingTimeInMin[1];
				lrPowerUV1_6 := fbAlfen6.stDataECS.lrTotalPower;	
					wStateUV1_6 := fbAlfen6.stDataECS.arrSocketStateECS[1];
						lrEnergySessionUV1_6 := fbAlfen6.stDataECS.arrSocketEnergySession[1];
							lrTotalEnergyUV1_6 := fbAlfen6.stDataECS.lrTotalCounterEnergy_Consumption;
	
(*---------------------------------------------CS7-----------------------------------------------------------*)	
	
//Manual Power
fbAlfen7.stSetupECS.bManualyOn := bManualyOnUV1_7;
	fbAlfen7.stSetupECS.byManualyTargetPower := byManualyTargetPowerUV1_7;
	
fbAlfen7(
	bEnable:= , 
	bPowerDataInvers:= , 
	byElectricFuseLine:= , 
	byUnitID_Socket1:= 1, 
	byUnitID_Socket2:= , 
	byNumberOfSockets:= 1, 
	byNumberOfConnectionWire:= 1, 
	diNrOfEMS_IN:= prgEMS.fbEMS.diNrOfEMS_OUT, 
	diNrOfEM_IN_CS:= , 
	sIPAdress:= '192.168.1.149',  
	stSetupECS:= , 
	stDataECS=> , 
	diNrOfECS_OUT=> );

bSManualyOn_UV1_7 := fbAlfen7.stDataECS.bSManualyOn;
	bySManualyTargetPowerUV1_7 := fbAlfen7.stDataECS.bySManualyTargetPower;	
		byErrorWarningUV1_7 := fbAlfen7.stDataECS.byErrorWarning;
			rChargingTimeInMinUV1_7 := fbAlfen7.stDataECS.arrChargingTimeInMin[1];
				lrPowerUV1_7 := fbAlfen7.stDataECS.lrTotalPower;	
					wStateUV1_7 := fbAlfen7.stDataECS.arrSocketStateECS[1];
						lrEnergySessionUV1_7 := fbAlfen7.stDataECS.arrSocketEnergySession[1];
							lrTotalEnergyUV1_7 := fbAlfen7.stDataECS.lrTotalCounterEnergy_Consumption;
	
(*---------------------------------------------CS8-----------------------------------------------------------*)	
	
//Manual Power
fbAlfen8.stSetupECS.bManualyOn := bManualyOnUV1_8;
	fbAlfen8.stSetupECS.byManualyTargetPower := byManualyTargetPowerUV1_8;
	
fbAlfen8(
	bEnable:= , 
	bPowerDataInvers:= , 
	byElectricFuseLine:= , 
	byUnitID_Socket1:= 1, 
	byUnitID_Socket2:= , 
	byNumberOfSockets:= 1, 
	byNumberOfConnectionWire:= 1, 
	diNrOfEMS_IN:= prgEMS.fbEMS.diNrOfEMS_OUT, 
	diNrOfEM_IN_CS:= , 
	sIPAdress:= '192.168.1.148',  
	stSetupECS:= , 
	stDataECS=> , 
	diNrOfECS_OUT=> );

bSManualyOn_UV1_8 := fbAlfen8.stDataECS.bSManualyOn;
	bySManualyTargetPowerUV1_8 := fbAlfen8.stDataECS.bySManualyTargetPower;	
		byErrorWarningUV1_8 := fbAlfen8.stDataECS.byErrorWarning;
			rChargingTimeInMinUV1_8 := fbAlfen8.stDataECS.arrChargingTimeInMin[1];
				lrPowerUV1_8 := fbAlfen8.stDataECS.lrTotalPower;	
					wStateUV1_8 := fbAlfen8.stDataECS.arrSocketStateECS[1];
						lrEnergySessionUV1_8 := fbAlfen8.stDataECS.arrSocketEnergySession[1];
							lrTotalEnergyUV1_8 := fbAlfen8.stDataECS.lrTotalCounterEnergy_Consumption;
	
(*---------------------------------------------CS9-----------------------------------------------------------*)	
	
//Manual Power
fbAlfen9.stSetupECS.bManualyOn := bManualyOnUV1_9;
	fbAlfen9.stSetupECS.byManualyTargetPower := byManualyTargetPowerUV1_9;
	
fbAlfen9(
	bEnable:= , 
	bPowerDataInvers:= , 
	byElectricFuseLine:= , 
	byUnitID_Socket1:= 1, 
	byUnitID_Socket2:= , 
	byNumberOfSockets:= 1, 
	byNumberOfConnectionWire:= 1, 
	diNrOfEMS_IN:= prgEMS.fbEMS.diNrOfEMS_OUT, 
	diNrOfEM_IN_CS:= , 
	sIPAdress:= '192.168.1.122',  
	stSetupECS:= , 
	stDataECS=> , 
	diNrOfECS_OUT=> );

bSManualyOn_UV1_9 := fbAlfen9.stDataECS.bSManualyOn;
	bySManualyTargetPowerUV1_9 := fbAlfen9.stDataECS.bySManualyTargetPower;
		byErrorWarningUV1_9 := fbAlfen9.stDataECS.byErrorWarning;	
			rChargingTimeInMinUV1_9 := fbAlfen9.stDataECS.arrChargingTimeInMin[1];
				lrPowerUV1_9 := fbAlfen9.stDataECS.lrTotalPower;	
					wStateUV1_9 := fbAlfen9.stDataECS.arrSocketStateECS[1];
						lrEnergySessionUV1_9 := fbAlfen9.stDataECS.arrSocketEnergySession[1];
							lrTotalEnergyUV1_9 := fbAlfen9.stDataECS.lrTotalCounterEnergy_Consumption;
	
(*---------------------------------------------CS10-----------------------------------------------------------*)	
	
//Manual Power
fbAlfen10.stSetupECS.bManualyOn := bManualyOnUV1_10;
	fbAlfen10.stSetupECS.byManualyTargetPower := byManualyTargetPowerUV1_10;
	
fbAlfen10(
	bEnable:= , 
	bPowerDataInvers:= , 
	byElectricFuseLine:= , 
	byUnitID_Socket1:= 1, 
	byUnitID_Socket2:= , 
	byNumberOfSockets:= 1, 
	byNumberOfConnectionWire:= 1, 
	diNrOfEMS_IN:= prgEMS.fbEMS.diNrOfEMS_OUT, 
	diNrOfEM_IN_CS:= , 
	sIPAdress:= '192.168.1.207', 
	stSetupECS:= , 
	stDataECS=> , 
	diNrOfECS_OUT=> );

bSManualyOn_UV1_10 := fbAlfen10.stDataECS.bSManualyOn;
	bySManualyTargetPowerUV1_10 := fbAlfen10.stDataECS.bySManualyTargetPower;
		byErrorWarningUV1_10 := fbAlfen10.stDataECS.byErrorWarning;	
			rChargingTimeInMinUV1_10 := fbAlfen10.stDataECS.arrChargingTimeInMin[1];
				lrPowerUV1_10 := fbAlfen10.stDataECS.lrTotalPower;	
					wStateUV1_10 := fbAlfen10.stDataECS.arrSocketStateECS[1];
						lrEnergySessionUV1_10 := fbAlfen10.stDataECS.arrSocketEnergySession[1];
							lrTotalEnergyUV1_10 := fbAlfen10.stDataECS.lrTotalCounterEnergy_Consumption;

END_PROGRAM

// ---- POUs/prgCS4.TcPOU
PROGRAM prgCS4
VAR
	fbAlfen1					: FB_ECS_Alfen_NG9xx_Platform;						//{#lynus.ag#()}
	fbAlfen2					: FB_ECS_Alfen_NG9xx_Platform;						//{#lynus.ag#()}
	fbAlfen3					: FB_ECS_Alfen_NG9xx_Platform;						//{#lynus.ag#()}
	fbAlfen4					: FB_ECS_Alfen_NG9xx_Platform;						//{#lynus.ag#()}
	fbAlfen5					: FB_ECS_Alfen_NG9xx_Platform;						//{#lynus.ag#()}
	fbAlfen6					: FB_ECS_Alfen_NG9xx_Platform;						//{#lynus.ag#()}
	fbAlfen7					: FB_ECS_Alfen_NG9xx_Platform;						//{#lynus.ag#()}
	fbAlfen8					: FB_ECS_Alfen_NG9xx_Platform;						//{#lynus.ag#()}
	fbAlfen9					: FB_ECS_Alfen_NG9xx_Platform;						//{#lynus.ag#()}
	fbAlfen10					: FB_ECS_Alfen_NG9xx_Platform;						//{#lynus.ag#()}
	
	bSManualyOn_UV1_1			: BOOL;												//{#lynus.ag#()}
	bySManualyTargetPowerUV1_1	: BYTE;												//{#lynus.ag#()}
	byErrorWarningUV1_1			: BYTE;												//{#lynus.ag#()}
	rChargingTimeInMinUV1_1		: REAL;												//{#lynus.ag#()}
	lrPowerUV1_1				: LREAL;											//{#lynus.ag#()}
	wStateUV1_1					: WORD;												//{#lynus.ag#()}
	lrEnergySessionUV1_1		: LREAL;											//{#lynus.ag#()}
	lrTotalEnergyUV1_1			: LREAL;											//{#lynus.ag#()}
	
	bSManualyOn_UV1_2			: BOOL;												//{#lynus.ag#()}
	bySManualyTargetPowerUV1_2	: BYTE;												//{#lynus.ag#()}
	byErrorWarningUV1_2			: BYTE;												//{#lynus.ag#()}
	rChargingTimeInMinUV1_2		: REAL;												//{#lynus.ag#()}
	lrPowerUV1_2				: LREAL;											//{#lynus.ag#()}
	wStateUV1_2					: WORD;												//{#lynus.ag#()}
	lrEnergySessionUV1_2		: LREAL;											//{#lynus.ag#()}
	lrTotalEnergyUV1_2			: LREAL;											//{#lynus.ag#()}
	
	bSManualyOn_UV1_3			: BOOL;												//{#lynus.ag#()}
	bySManualyTargetPowerUV1_3	: BYTE;												//{#lynus.ag#()}
	byErrorWarningUV1_3			: BYTE;												//{#lynus.ag#()}
	rChargingTimeInMinUV1_3		: REAL;												//{#lynus.ag#()}
	lrPowerUV1_3				: LREAL;											//{#lynus.ag#()}
	wStateUV1_3					: WORD;												//{#lynus.ag#()}
	lrEnergySessionUV1_3		: LREAL;											//{#lynus.ag#()}
	lrTotalEnergyUV1_3			: LREAL;											//{#lynus.ag#()}
	
	bSManualyOn_UV1_4			: BOOL;												//{#lynus.ag#()}
	bySManualyTargetPowerUV1_4	: BYTE;												//{#lynus.ag#()}
	byErrorWarningUV1_4			: BYTE;												//{#lynus.ag#()}
	rChargingTimeInMinUV1_4		: REAL;												//{#lynus.ag#()}
	lrPowerUV1_4				: LREAL;											//{#lynus.ag#()}
	wStateUV1_4					: WORD;												//{#lynus.ag#()}
	lrEnergySessionUV1_4		: LREAL;											//{#lynus.ag#()}
	lrTotalEnergyUV1_4			: LREAL;											//{#lynus.ag#()}
	
	bSManualyOn_UV1_5			: BOOL;												//{#lynus.ag#()}
	bySManualyTargetPowerUV1_5	: BYTE;												//{#lynus.ag#()}
	byErrorWarningUV1_5			: BYTE;												//{#lynus.ag#()}
	rChargingTimeInMinUV1_5		: REAL;												//{#lynus.ag#()}
	lrPowerUV1_5				: LREAL;											//{#lynus.ag#()}
	wStateUV1_5					: WORD;												//{#lynus.ag#()}
	lrEnergySessionUV1_5		: LREAL;											//{#lynus.ag#()}
	lrTotalEnergyUV1_5			: LREAL;											//{#lynus.ag#()}
	
	bSManualyOn_UV1_6			: BOOL;												//{#lynus.ag#()}
	bySManualyTargetPowerUV1_6	: BYTE;												//{#lynus.ag#()}
	byErrorWarningUV1_6			: BYTE;												//{#lynus.ag#()}
	rChargingTimeInMinUV1_6		: REAL;												//{#lynus.ag#()}
	lrPowerUV1_6				: LREAL;											//{#lynus.ag#()}
	wStateUV1_6					: WORD;												//{#lynus.ag#()}
	lrEnergySessionUV1_6		: LREAL;											//{#lynus.ag#()}
	lrTotalEnergyUV1_6			: LREAL;											//{#lynus.ag#()}
	
	bSManualyOn_UV1_7			: BOOL;												//{#lynus.ag#()}
	bySManualyTargetPowerUV1_7	: BYTE;												//{#lynus.ag#()}
	byErrorWarningUV1_7			: BYTE;												//{#lynus.ag#()}
	rChargingTimeInMinUV1_7		: REAL;												//{#lynus.ag#()}
	lrPowerUV1_7				: LREAL;											//{#lynus.ag#()}
	wStateUV1_7					: WORD;												//{#lynus.ag#()}
	lrEnergySessionUV1_7		: LREAL;											//{#lynus.ag#()}
	lrTotalEnergyUV1_7			: LREAL;											//{#lynus.ag#()}
	
	bSManualyOn_UV1_8			: BOOL;												//{#lynus.ag#()}
	bySManualyTargetPowerUV1_8	: BYTE;												//{#lynus.ag#()}
	byErrorWarningUV1_8			: BYTE;												//{#lynus.ag#()}
	rChargingTimeInMinUV1_8		: REAL;												//{#lynus.ag#()}
	lrPowerUV1_8				: LREAL;											//{#lynus.ag#()}
	wStateUV1_8					: WORD;												//{#lynus.ag#()}
	lrEnergySessionUV1_8		: LREAL;											//{#lynus.ag#()}
	lrTotalEnergyUV1_8			: LREAL;											//{#lynus.ag#()}
	
	bSManualyOn_UV1_9			: BOOL;												//{#lynus.ag#()}
	bySManualyTargetPowerUV1_9	: BYTE;												//{#lynus.ag#()}
	byErrorWarningUV1_9			: BYTE;												//{#lynus.ag#()}
	rChargingTimeInMinUV1_9		: REAL;												//{#lynus.ag#()}
	lrPowerUV1_9				: LREAL;											//{#lynus.ag#()}
	wStateUV1_9					: WORD;												//{#lynus.ag#()}
	lrEnergySessionUV1_9		: LREAL;											//{#lynus.ag#()}
	lrTotalEnergyUV1_9			: LREAL;											//{#lynus.ag#()}
	
	bSManualyOn_UV1_10			: BOOL;												//{#lynus.ag#()}
	bySManualyTargetPowerUV1_10	: BYTE;												//{#lynus.ag#()}
	byErrorWarningUV1_10		: BYTE;												//{#lynus.ag#()}
	rChargingTimeInMinUV1_10	: REAL;												//{#lynus.ag#()}
	lrPowerUV1_10				: LREAL;											//{#lynus.ag#()}
	wStateUV1_10				: WORD;												//{#lynus.ag#()}
	lrEnergySessionUV1_10		: LREAL;											//{#lynus.ag#()}
	lrTotalEnergyUV1_10			: LREAL;											//{#lynus.ag#()}
END_VAR
VAR PERSISTENT
	bManualyOnUV1_1				: BOOL;												//{#lynus.ag#()}
	byManualyTargetPowerUV1_1	: BYTE;												//{#lynus.ag#()}
	
	bManualyOnUV1_2				: BOOL;												//{#lynus.ag#()}
	byManualyTargetPowerUV1_2	: BYTE;												//{#lynus.ag#()}
	
	bManualyOnUV1_3				: BOOL;												//{#lynus.ag#()}
	byManualyTargetPowerUV1_3	: BYTE;												//{#lynus.ag#()}
	
	bManualyOnUV1_4				: BOOL;												//{#lynus.ag#()}
	byManualyTargetPowerUV1_4	: BYTE;												//{#lynus.ag#()}
	
	bManualyOnUV1_5				: BOOL;												//{#lynus.ag#()}
	byManualyTargetPowerUV1_5	: BYTE;												//{#lynus.ag#()}
	
	bManualyOnUV1_6				: BOOL;												//{#lynus.ag#()}
	byManualyTargetPowerUV1_6	: BYTE;												//{#lynus.ag#()}
	
	bManualyOnUV1_7				: BOOL;												//{#lynus.ag#()}
	byManualyTargetPowerUV1_7	: BYTE;												//{#lynus.ag#()}
	
	bManualyOnUV1_8				: BOOL;												//{#lynus.ag#()}
	byManualyTargetPowerUV1_8	: BYTE;												//{#lynus.ag#()}
	
	bManualyOnUV1_9				: BOOL;												//{#lynus.ag#()}
	byManualyTargetPowerUV1_9	: BYTE;												//{#lynus.ag#()}
	
	bManualyOnUV1_10			: BOOL;												//{#lynus.ag#()}
	byManualyTargetPowerUV1_10	: BYTE;												//{#lynus.ag#()}
END_VAR

(*---------------------------------------------CS1-----------------------------------------------------------*)

//Manual Power
fbAlfen1.stSetupECS.bManualyOn := bManualyOnUV1_1;
	fbAlfen1.stSetupECS.byManualyTargetPower := byManualyTargetPowerUV1_1;

fbAlfen1(
	bEnable:= , 
	bPowerDataInvers:= , 
	byElectricFuseLine:= , 
	byUnitID_Socket1:= 1, 
	byUnitID_Socket2:= , 
	byNumberOfSockets:= 1, 
	byNumberOfConnectionWire:= 1, 
	diNrOfEMS_IN:= prgEMS.fbEMS.diNrOfEMS_OUT, 
	diNrOfEM_IN_CS:= , 
	sIPAdress:= '192.168.1.243', 
	stSetupECS:= , 
	stDataECS=> , 
	diNrOfECS_OUT=> );

bSManualyOn_UV1_1 := fbAlfen1.stDataECS.bSManualyOn;
	bySManualyTargetPowerUV1_1 := fbAlfen1.stDataECS.bySManualyTargetPower;
		byErrorWarningUV1_1 := fbAlfen1.stDataECS.byErrorWarning;	
			rChargingTimeInMinUV1_1 := fbAlfen1.stDataECS.arrChargingTimeInMin[1];
				lrPowerUV1_1 := fbAlfen1.stDataECS.lrTotalPower;	
					wStateUV1_1 := fbAlfen1.stDataECS.arrSocketStateECS[1];
						lrEnergySessionUV1_1 := fbAlfen1.stDataECS.arrSocketEnergySession[1];
							lrTotalEnergyUV1_1 := fbAlfen1.stDataECS.lrTotalCounterEnergy_Consumption;	
	
(*---------------------------------------------CS2-----------------------------------------------------------*)
	
//Manual Power
fbAlfen2.stSetupECS.bManualyOn := bManualyOnUV1_2;
	fbAlfen2.stSetupECS.byManualyTargetPower := byManualyTargetPowerUV1_2;
	
fbAlfen2(
	bEnable:= , 
	bPowerDataInvers:= , 
	byElectricFuseLine:= , 
	byUnitID_Socket1:= 1, 
	byUnitID_Socket2:= , 
	byNumberOfSockets:= 1, 
	byNumberOfConnectionWire:= 1, 
	diNrOfEMS_IN:= prgEMS.fbEMS.diNrOfEMS_OUT, 
	diNrOfEM_IN_CS:= , 
	sIPAdress:= '192.168.1.200', 
	stSetupECS:= , 
	stDataECS=> , 
	diNrOfECS_OUT=> );

bSManualyOn_UV1_2 := fbAlfen2.stDataECS.bSManualyOn;
	bySManualyTargetPowerUV1_2 := fbAlfen2.stDataECS.bySManualyTargetPower;	
		byErrorWarningUV1_2 := fbAlfen2.stDataECS.byErrorWarning;
			rChargingTimeInMinUV1_2 := fbAlfen2.stDataECS.arrChargingTimeInMin[1];;
				lrPowerUV1_2 := fbAlfen2.stDataECS.lrTotalPower;	
					wStateUV1_2 := fbAlfen2.stDataECS.arrSocketStateECS[1];
						lrEnergySessionUV1_2 := fbAlfen2.stDataECS.arrSocketEnergySession[1];
							lrTotalEnergyUV1_2 := fbAlfen2.stDataECS.lrTotalCounterEnergy_Consumption;
	
(*---------------------------------------------CS3-----------------------------------------------------------*)	
	
//Manual Power
fbAlfen3.stSetupECS.bManualyOn := bManualyOnUV1_3;
	fbAlfen3.stSetupECS.byManualyTargetPower := byManualyTargetPowerUV1_3;
	
fbAlfen3(
	bEnable:= , 
	bPowerDataInvers:= , 
	byElectricFuseLine:= , 
	byUnitID_Socket1:= 1, 
	byUnitID_Socket2:= , 
	byNumberOfSockets:= 1, 
	byNumberOfConnectionWire:= 1, 
	diNrOfEMS_IN:= prgEMS.fbEMS.diNrOfEMS_OUT, 
	diNrOfEM_IN_CS:= , 
	sIPAdress:= '192.168.1.172',  
	stSetupECS:= , 
	stDataECS=> , 
	diNrOfECS_OUT=> );

bSManualyOn_UV1_3 := fbAlfen3.stDataECS.bSManualyOn;
	bySManualyTargetPowerUV1_3 := fbAlfen3.stDataECS.bySManualyTargetPower;
		byErrorWarningUV1_3 := fbAlfen3.stDataECS.byErrorWarning;
			rChargingTimeInMinUV1_3 := fbAlfen3.stDataECS.arrChargingTimeInMin[1];	
				lrPowerUV1_3 := fbAlfen3.stDataECS.lrTotalPower;	
					wStateUV1_3 := fbAlfen3.stDataECS.arrSocketStateECS[1];
						lrEnergySessionUV1_3 := fbAlfen3.stDataECS.arrSocketEnergySession[1];
							lrTotalEnergyUV1_3 := fbAlfen3.stDataECS.lrTotalCounterEnergy_Consumption;		
	
(*---------------------------------------------CS4-----------------------------------------------------------*)	
	
//Manual Power
fbAlfen4.stSetupECS.bManualyOn := bManualyOnUV1_4;
	fbAlfen4.stSetupECS.byManualyTargetPower := byManualyTargetPowerUV1_4;
	
fbAlfen4(
	bEnable:= , 
	bPowerDataInvers:= , 
	byElectricFuseLine:= , 
	byUnitID_Socket1:= 1, 
	byUnitID_Socket2:= , 
	byNumberOfSockets:= 1, 
	byNumberOfConnectionWire:= 1, 
	diNrOfEMS_IN:= prgEMS.fbEMS.diNrOfEMS_OUT, 
	diNrOfEM_IN_CS:= , 
	sIPAdress:= '192.168.1.142',  
	stSetupECS:= , 
	stDataECS=> , 
	diNrOfECS_OUT=> );

bSManualyOn_UV1_4 := fbAlfen4.stDataECS.bSManualyOn;
	bySManualyTargetPowerUV1_4 := fbAlfen4.stDataECS.bySManualyTargetPower;	
		byErrorWarningUV1_4 := fbAlfen4.stDataECS.byErrorWarning;
			rChargingTimeInMinUV1_4 := fbAlfen4.stDataECS.arrChargingTimeInMin[1];
				lrPowerUV1_4 := fbAlfen4.stDataECS.lrTotalPower;	
					wStateUV1_4 := fbAlfen4.stDataECS.arrSocketStateECS[1];
						lrEnergySessionUV1_4 := fbAlfen4.stDataECS.arrSocketEnergySession[1];
							lrTotalEnergyUV1_4 := fbAlfen4.stDataECS.lrTotalCounterEnergy_Consumption;
	
(*---------------------------------------------CS5-----------------------------------------------------------*)	
	
//Manual Power
fbAlfen5.stSetupECS.bManualyOn := bManualyOnUV1_5;
	fbAlfen5.stSetupECS.byManualyTargetPower := byManualyTargetPowerUV1_5;
	
fbAlfen5(
	bEnable:= , 
	bPowerDataInvers:= , 
	byElectricFuseLine:= , 
	byUnitID_Socket1:= 1, 
	byUnitID_Socket2:= , 
	byNumberOfSockets:= 1, 
	byNumberOfConnectionWire:= 1, 
	diNrOfEMS_IN:= prgEMS.fbEMS.diNrOfEMS_OUT, 
	diNrOfEM_IN_CS:= , 
	sIPAdress:= '192.168.1.136',  
	stSetupECS:= , 
	stDataECS=> , 
	diNrOfECS_OUT=> );

bSManualyOn_UV1_5 := fbAlfen5.stDataECS.bSManualyOn;
	bySManualyTargetPowerUV1_5 := fbAlfen5.stDataECS.bySManualyTargetPower;
		byErrorWarningUV1_5 := fbAlfen5.stDataECS.byErrorWarning;
			rChargingTimeInMinUV1_5 := fbAlfen5.stDataECS.arrChargingTimeInMin[1];
				lrPowerUV1_5 := fbAlfen5.stDataECS.lrTotalPower;	
					wStateUV1_5 := fbAlfen5.stDataECS.arrSocketStateECS[1];
						lrEnergySessionUV1_5 := fbAlfen5.stDataECS.arrSocketEnergySession[1];
							lrTotalEnergyUV1_5 := fbAlfen5.stDataECS.lrTotalCounterEnergy_Consumption;		
	
(*---------------------------------------------CS6-----------------------------------------------------------*)	
	
//Manual Power
fbAlfen6.stSetupECS.bManualyOn := bManualyOnUV1_6;
	fbAlfen6.stSetupECS.byManualyTargetPower := byManualyTargetPowerUV1_6;
	
fbAlfen6(
	bEnable:= , 
	bPowerDataInvers:= , 
	byElectricFuseLine:= , 
	byUnitID_Socket1:= 1, 
	byUnitID_Socket2:= , 
	byNumberOfSockets:= 1, 
	byNumberOfConnectionWire:= 1, 
	diNrOfEMS_IN:= prgEMS.fbEMS.diNrOfEMS_OUT, 
	diNrOfEM_IN_CS:= , 
	sIPAdress:= '192.168.1.232',  
	stSetupECS:= , 
	stDataECS=> , 
	diNrOfECS_OUT=> );

bSManualyOn_UV1_6 := fbAlfen6.stDataECS.bSManualyOn;
	bySManualyTargetPowerUV1_6 := fbAlfen6.stDataECS.bySManualyTargetPower;	
		byErrorWarningUV1_6 := fbAlfen6.stDataECS.byErrorWarning;
			rChargingTimeInMinUV1_6 := fbAlfen6.stDataECS.arrChargingTimeInMin[1];
				lrPowerUV1_6 := fbAlfen6.stDataECS.lrTotalPower;	
					wStateUV1_6 := fbAlfen6.stDataECS.arrSocketStateECS[1];
						lrEnergySessionUV1_6 := fbAlfen6.stDataECS.arrSocketEnergySession[1];
							lrTotalEnergyUV1_6 := fbAlfen6.stDataECS.lrTotalCounterEnergy_Consumption;
	
(*---------------------------------------------CS7-----------------------------------------------------------*)	
	
//Manual Power
fbAlfen7.stSetupECS.bManualyOn := bManualyOnUV1_7;
	fbAlfen7.stSetupECS.byManualyTargetPower := byManualyTargetPowerUV1_7;
	
fbAlfen7(
	bEnable:= , 
	bPowerDataInvers:= , 
	byElectricFuseLine:= , 
	byUnitID_Socket1:= 1, 
	byUnitID_Socket2:= , 
	byNumberOfSockets:= 1, 
	byNumberOfConnectionWire:= 1, 
	diNrOfEMS_IN:= prgEMS.fbEMS.diNrOfEMS_OUT, 
	diNrOfEM_IN_CS:= , 
	sIPAdress:= '192.168.1.193',  
	stSetupECS:= , 
	stDataECS=> , 
	diNrOfECS_OUT=> );

bSManualyOn_UV1_7 := fbAlfen7.stDataECS.bSManualyOn;
	bySManualyTargetPowerUV1_7 := fbAlfen7.stDataECS.bySManualyTargetPower;	
		byErrorWarningUV1_7 := fbAlfen7.stDataECS.byErrorWarning;
			rChargingTimeInMinUV1_7 := fbAlfen7.stDataECS.arrChargingTimeInMin[1];
				lrPowerUV1_7 := fbAlfen7.stDataECS.lrTotalPower;	
					wStateUV1_7 := fbAlfen7.stDataECS.arrSocketStateECS[1];
						lrEnergySessionUV1_7 := fbAlfen7.stDataECS.arrSocketEnergySession[1];
							lrTotalEnergyUV1_7 := fbAlfen7.stDataECS.lrTotalCounterEnergy_Consumption;
	
(*---------------------------------------------CS8-----------------------------------------------------------*)	
	
//Manual Power
fbAlfen8.stSetupECS.bManualyOn := bManualyOnUV1_8;
	fbAlfen8.stSetupECS.byManualyTargetPower := byManualyTargetPowerUV1_8;
	
fbAlfen8(
	bEnable:= , 
	bPowerDataInvers:= , 
	byElectricFuseLine:= , 
	byUnitID_Socket1:= 1, 
	byUnitID_Socket2:= , 
	byNumberOfSockets:= 1, 
	byNumberOfConnectionWire:= 1, 
	diNrOfEMS_IN:= prgEMS.fbEMS.diNrOfEMS_OUT, 
	diNrOfEM_IN_CS:= , 
	sIPAdress:= '192.168.1.102',  
	stSetupECS:= , 
	stDataECS=> , 
	diNrOfECS_OUT=> );

bSManualyOn_UV1_8 := fbAlfen8.stDataECS.bSManualyOn;
	bySManualyTargetPowerUV1_8 := fbAlfen8.stDataECS.bySManualyTargetPower;	
		byErrorWarningUV1_8 := fbAlfen8.stDataECS.byErrorWarning;
			rChargingTimeInMinUV1_8 := fbAlfen8.stDataECS.arrChargingTimeInMin[1];
				lrPowerUV1_8 := fbAlfen8.stDataECS.lrTotalPower;	
					wStateUV1_8 := fbAlfen8.stDataECS.arrSocketStateECS[1];
						lrEnergySessionUV1_8 := fbAlfen8.stDataECS.arrSocketEnergySession[1];
							lrTotalEnergyUV1_8 := fbAlfen8.stDataECS.lrTotalCounterEnergy_Consumption;
	
(*---------------------------------------------CS9-----------------------------------------------------------*)	
	
//Manual Power
fbAlfen9.stSetupECS.bManualyOn := bManualyOnUV1_9;
	fbAlfen9.stSetupECS.byManualyTargetPower := byManualyTargetPowerUV1_9;
	
fbAlfen9(
	bEnable:= , 
	bPowerDataInvers:= , 
	byElectricFuseLine:= , 
	byUnitID_Socket1:= 1, 
	byUnitID_Socket2:= , 
	byNumberOfSockets:= 1, 
	byNumberOfConnectionWire:= 1, 
	diNrOfEMS_IN:= prgEMS.fbEMS.diNrOfEMS_OUT, 
	diNrOfEM_IN_CS:= , 
	sIPAdress:= '192.168.1.240',  
	stSetupECS:= , 
	stDataECS=> , 
	diNrOfECS_OUT=> );

bSManualyOn_UV1_9 := fbAlfen9.stDataECS.bSManualyOn;
	bySManualyTargetPowerUV1_9 := fbAlfen9.stDataECS.bySManualyTargetPower;
		byErrorWarningUV1_9 := fbAlfen9.stDataECS.byErrorWarning;	
			rChargingTimeInMinUV1_9 := fbAlfen9.stDataECS.arrChargingTimeInMin[1];
				lrPowerUV1_9 := fbAlfen9.stDataECS.lrTotalPower;	
					wStateUV1_9 := fbAlfen9.stDataECS.arrSocketStateECS[1];
						lrEnergySessionUV1_9 := fbAlfen9.stDataECS.arrSocketEnergySession[1];
							lrTotalEnergyUV1_9 := fbAlfen9.stDataECS.lrTotalCounterEnergy_Consumption;
	
(*---------------------------------------------CS10-----------------------------------------------------------*)	
	
//Manual Power
fbAlfen10.stSetupECS.bManualyOn := bManualyOnUV1_10;
	fbAlfen10.stSetupECS.byManualyTargetPower := byManualyTargetPowerUV1_10;
	
fbAlfen10(
	bEnable:= , 
	bPowerDataInvers:= , 
	byElectricFuseLine:= , 
	byUnitID_Socket1:= 1, 
	byUnitID_Socket2:= , 
	byNumberOfSockets:= 1, 
	byNumberOfConnectionWire:= 1, 
	diNrOfEMS_IN:= prgEMS.fbEMS.diNrOfEMS_OUT, 
	diNrOfEM_IN_CS:= , 
	sIPAdress:= '192.168.1.173', 
	stSetupECS:= , 
	stDataECS=> , 
	diNrOfECS_OUT=> );

bSManualyOn_UV1_10 := fbAlfen10.stDataECS.bSManualyOn;
	bySManualyTargetPowerUV1_10 := fbAlfen10.stDataECS.bySManualyTargetPower;
		byErrorWarningUV1_10 := fbAlfen10.stDataECS.byErrorWarning;	
			rChargingTimeInMinUV1_10 := fbAlfen10.stDataECS.arrChargingTimeInMin[1];
				lrPowerUV1_10 := fbAlfen10.stDataECS.lrTotalPower;	
					wStateUV1_10 := fbAlfen10.stDataECS.arrSocketStateECS[1];
						lrEnergySessionUV1_10 := fbAlfen10.stDataECS.arrSocketEnergySession[1];
							lrTotalEnergyUV1_10 := fbAlfen10.stDataECS.lrTotalCounterEnergy_Consumption;

END_PROGRAM

// ---- POUs/prgCS5.TcPOU
PROGRAM prgCS5
VAR
	fbAlfen1					: FB_ECS_Alfen_NG9xx_Platform;						//{#lynus.ag#()}
	fbAlfen2					: FB_ECS_Alfen_NG9xx_Platform;						//{#lynus.ag#()}
	fbAlfen3					: FB_ECS_Alfen_NG9xx_Platform;						//{#lynus.ag#()}
	fbAlfen4					: FB_ECS_Alfen_NG9xx_Platform;						//{#lynus.ag#()}
	fbAlfen5					: FB_ECS_Alfen_NG9xx_Platform;						//{#lynus.ag#()}
	fbAlfen6					: FB_ECS_Alfen_NG9xx_Platform;						//{#lynus.ag#()}
	fbAlfen7					: FB_ECS_Alfen_NG9xx_Platform;						//{#lynus.ag#()}
	fbAlfen8					: FB_ECS_Alfen_NG9xx_Platform;						//{#lynus.ag#()}
	fbAlfen9					: FB_ECS_Alfen_NG9xx_Platform;						//{#lynus.ag#()}
	fbAlfen10					: FB_ECS_Alfen_NG9xx_Platform;						//{#lynus.ag#()}
	
	bSManualyOn_UV1_1			: BOOL;												//{#lynus.ag#()}
	bySManualyTargetPowerUV1_1	: BYTE;												//{#lynus.ag#()}
	byErrorWarningUV1_1			: BYTE;												//{#lynus.ag#()}
	rChargingTimeInMinUV1_1		: REAL;												//{#lynus.ag#()}
	lrPowerUV1_1				: LREAL;											//{#lynus.ag#()}
	wStateUV1_1					: WORD;												//{#lynus.ag#()}
	lrEnergySessionUV1_1		: LREAL;											//{#lynus.ag#()}
	lrTotalEnergyUV1_1			: LREAL;											//{#lynus.ag#()}
	
	bSManualyOn_UV1_2			: BOOL;												//{#lynus.ag#()}
	bySManualyTargetPowerUV1_2	: BYTE;												//{#lynus.ag#()}
	byErrorWarningUV1_2			: BYTE;												//{#lynus.ag#()}
	rChargingTimeInMinUV1_2		: REAL;												//{#lynus.ag#()}
	lrPowerUV1_2				: LREAL;											//{#lynus.ag#()}
	wStateUV1_2					: WORD;												//{#lynus.ag#()}
	lrEnergySessionUV1_2		: LREAL;											//{#lynus.ag#()}
	lrTotalEnergyUV1_2			: LREAL;											//{#lynus.ag#()}
	
	bSManualyOn_UV1_3			: BOOL;												//{#lynus.ag#()}
	bySManualyTargetPowerUV1_3	: BYTE;												//{#lynus.ag#()}
	byErrorWarningUV1_3			: BYTE;												//{#lynus.ag#()}
	rChargingTimeInMinUV1_3		: REAL;												//{#lynus.ag#()}
	lrPowerUV1_3				: LREAL;											//{#lynus.ag#()}
	wStateUV1_3					: WORD;												//{#lynus.ag#()}
	lrEnergySessionUV1_3		: LREAL;											//{#lynus.ag#()}
	lrTotalEnergyUV1_3			: LREAL;											//{#lynus.ag#()}
	
	bSManualyOn_UV1_4			: BOOL;												//{#lynus.ag#()}
	bySManualyTargetPowerUV1_4	: BYTE;												//{#lynus.ag#()}
	byErrorWarningUV1_4			: BYTE;												//{#lynus.ag#()}
	rChargingTimeInMinUV1_4		: REAL;												//{#lynus.ag#()}
	lrPowerUV1_4				: LREAL;											//{#lynus.ag#()}
	wStateUV1_4					: WORD;												//{#lynus.ag#()}
	lrEnergySessionUV1_4		: LREAL;											//{#lynus.ag#()}
	lrTotalEnergyUV1_4			: LREAL;											//{#lynus.ag#()}
	
	bSManualyOn_UV1_5			: BOOL;												//{#lynus.ag#()}
	bySManualyTargetPowerUV1_5	: BYTE;												//{#lynus.ag#()}
	byErrorWarningUV1_5			: BYTE;												//{#lynus.ag#()}
	rChargingTimeInMinUV1_5		: REAL;												//{#lynus.ag#()}
	lrPowerUV1_5				: LREAL;											//{#lynus.ag#()}
	wStateUV1_5					: WORD;												//{#lynus.ag#()}
	lrEnergySessionUV1_5		: LREAL;											//{#lynus.ag#()}
	lrTotalEnergyUV1_5			: LREAL;											//{#lynus.ag#()}
	
	bSManualyOn_UV1_6			: BOOL;												//{#lynus.ag#()}
	bySManualyTargetPowerUV1_6	: BYTE;												//{#lynus.ag#()}
	byErrorWarningUV1_6			: BYTE;												//{#lynus.ag#()}
	rChargingTimeInMinUV1_6		: REAL;												//{#lynus.ag#()}
	lrPowerUV1_6				: LREAL;											//{#lynus.ag#()}
	wStateUV1_6					: WORD;												//{#lynus.ag#()}
	lrEnergySessionUV1_6		: LREAL;											//{#lynus.ag#()}
	lrTotalEnergyUV1_6			: LREAL;											//{#lynus.ag#()}
	
	bSManualyOn_UV1_7			: BOOL;												//{#lynus.ag#()}
	bySManualyTargetPowerUV1_7	: BYTE;												//{#lynus.ag#()}
	byErrorWarningUV1_7			: BYTE;												//{#lynus.ag#()}
	rChargingTimeInMinUV1_7		: REAL;												//{#lynus.ag#()}
	lrPowerUV1_7				: LREAL;											//{#lynus.ag#()}
	wStateUV1_7					: WORD;												//{#lynus.ag#()}
	lrEnergySessionUV1_7		: LREAL;											//{#lynus.ag#()}
	lrTotalEnergyUV1_7			: LREAL;											//{#lynus.ag#()}
	
	bSManualyOn_UV1_8			: BOOL;												//{#lynus.ag#()}
	bySManualyTargetPowerUV1_8	: BYTE;												//{#lynus.ag#()}
	byErrorWarningUV1_8			: BYTE;												//{#lynus.ag#()}
	rChargingTimeInMinUV1_8		: REAL;												//{#lynus.ag#()}
	lrPowerUV1_8				: LREAL;											//{#lynus.ag#()}
	wStateUV1_8					: WORD;												//{#lynus.ag#()}
	lrEnergySessionUV1_8		: LREAL;											//{#lynus.ag#()}
	lrTotalEnergyUV1_8			: LREAL;											//{#lynus.ag#()}
	
	bSManualyOn_UV1_9			: BOOL;												//{#lynus.ag#()}
	bySManualyTargetPowerUV1_9	: BYTE;												//{#lynus.ag#()}
	byErrorWarningUV1_9			: BYTE;												//{#lynus.ag#()}
	rChargingTimeInMinUV1_9		: REAL;												//{#lynus.ag#()}
	lrPowerUV1_9				: LREAL;											//{#lynus.ag#()}
	wStateUV1_9					: WORD;												//{#lynus.ag#()}
	lrEnergySessionUV1_9		: LREAL;											//{#lynus.ag#()}
	lrTotalEnergyUV1_9			: LREAL;											//{#lynus.ag#()}
	
	bSManualyOn_UV1_10			: BOOL;												//{#lynus.ag#()}
	bySManualyTargetPowerUV1_10	: BYTE;												//{#lynus.ag#()}
	byErrorWarningUV1_10		: BYTE;												//{#lynus.ag#()}
	rChargingTimeInMinUV1_10	: REAL;												//{#lynus.ag#()}
	lrPowerUV1_10				: LREAL;											//{#lynus.ag#()}
	wStateUV1_10				: WORD;												//{#lynus.ag#()}
	lrEnergySessionUV1_10		: LREAL;											//{#lynus.ag#()}
	lrTotalEnergyUV1_10			: LREAL;											//{#lynus.ag#()}
END_VAR
VAR PERSISTENT
	bManualyOnUV1_1				: BOOL;												//{#lynus.ag#()}
	byManualyTargetPowerUV1_1	: BYTE;												//{#lynus.ag#()}
	
	bManualyOnUV1_2				: BOOL;												//{#lynus.ag#()}
	byManualyTargetPowerUV1_2	: BYTE;												//{#lynus.ag#()}
	
	bManualyOnUV1_3				: BOOL;												//{#lynus.ag#()}
	byManualyTargetPowerUV1_3	: BYTE;												//{#lynus.ag#()}
	
	bManualyOnUV1_4				: BOOL;												//{#lynus.ag#()}
	byManualyTargetPowerUV1_4	: BYTE;												//{#lynus.ag#()}
	
	bManualyOnUV1_5				: BOOL;												//{#lynus.ag#()}
	byManualyTargetPowerUV1_5	: BYTE;												//{#lynus.ag#()}
	
	bManualyOnUV1_6				: BOOL;												//{#lynus.ag#()}
	byManualyTargetPowerUV1_6	: BYTE;												//{#lynus.ag#()}
	
	bManualyOnUV1_7				: BOOL;												//{#lynus.ag#()}
	byManualyTargetPowerUV1_7	: BYTE;												//{#lynus.ag#()}
	
	bManualyOnUV1_8				: BOOL;												//{#lynus.ag#()}
	byManualyTargetPowerUV1_8	: BYTE;												//{#lynus.ag#()}
	
	bManualyOnUV1_9				: BOOL;												//{#lynus.ag#()}
	byManualyTargetPowerUV1_9	: BYTE;												//{#lynus.ag#()}
	
	bManualyOnUV1_10			: BOOL;												//{#lynus.ag#()}
	byManualyTargetPowerUV1_10	: BYTE;												//{#lynus.ag#()}
END_VAR

(*---------------------------------------------CS1-----------------------------------------------------------*)

//Manual Power
fbAlfen1.stSetupECS.bManualyOn := bManualyOnUV1_1;
	fbAlfen1.stSetupECS.byManualyTargetPower := byManualyTargetPowerUV1_1;

fbAlfen1(
	bEnable:= , 
	bPowerDataInvers:= , 
	byElectricFuseLine:= , 
	byUnitID_Socket1:= 1, 
	byUnitID_Socket2:= , 
	byNumberOfSockets:= 1, 
	byNumberOfConnectionWire:= 1, 
	diNrOfEMS_IN:= prgEMS.fbEMS.diNrOfEMS_OUT, 
	diNrOfEM_IN_CS:= , 
	sIPAdress:= '192.168.1.138', 
	stSetupECS:= , 
	stDataECS=> , 
	diNrOfECS_OUT=> );

bSManualyOn_UV1_1 := fbAlfen1.stDataECS.bSManualyOn;
	bySManualyTargetPowerUV1_1 := fbAlfen1.stDataECS.bySManualyTargetPower;
		byErrorWarningUV1_1 := fbAlfen1.stDataECS.byErrorWarning;	
			rChargingTimeInMinUV1_1 := fbAlfen1.stDataECS.arrChargingTimeInMin[1];
				lrPowerUV1_1 := fbAlfen1.stDataECS.lrTotalPower;	
					wStateUV1_1 := fbAlfen1.stDataECS.arrSocketStateECS[1];
						lrEnergySessionUV1_1 := fbAlfen1.stDataECS.arrSocketEnergySession[1];
							lrTotalEnergyUV1_1 := fbAlfen1.stDataECS.lrTotalCounterEnergy_Consumption;	
	
(*---------------------------------------------CS2-----------------------------------------------------------*)
	
//Manual Power
fbAlfen2.stSetupECS.bManualyOn := bManualyOnUV1_2;
	fbAlfen2.stSetupECS.byManualyTargetPower := byManualyTargetPowerUV1_2;
	
fbAlfen2(
	bEnable:= , 
	bPowerDataInvers:= , 
	byElectricFuseLine:= , 
	byUnitID_Socket1:= 1, 
	byUnitID_Socket2:= , 
	byNumberOfSockets:= 1, 
	byNumberOfConnectionWire:= 1, 
	diNrOfEMS_IN:= prgEMS.fbEMS.diNrOfEMS_OUT, 
	diNrOfEM_IN_CS:= , 
	sIPAdress:= '192.168.1.239', 
	stSetupECS:= , 
	stDataECS=> , 
	diNrOfECS_OUT=> );

bSManualyOn_UV1_2 := fbAlfen2.stDataECS.bSManualyOn;
	bySManualyTargetPowerUV1_2 := fbAlfen2.stDataECS.bySManualyTargetPower;	
		byErrorWarningUV1_2 := fbAlfen2.stDataECS.byErrorWarning;
			rChargingTimeInMinUV1_2 := fbAlfen2.stDataECS.arrChargingTimeInMin[1];;
				lrPowerUV1_2 := fbAlfen2.stDataECS.lrTotalPower;	
					wStateUV1_2 := fbAlfen2.stDataECS.arrSocketStateECS[1];
						lrEnergySessionUV1_2 := fbAlfen2.stDataECS.arrSocketEnergySession[1];
							lrTotalEnergyUV1_2 := fbAlfen2.stDataECS.lrTotalCounterEnergy_Consumption;
	
(*---------------------------------------------CS3-----------------------------------------------------------*)	
	
//Manual Power
fbAlfen3.stSetupECS.bManualyOn := bManualyOnUV1_3;
	fbAlfen3.stSetupECS.byManualyTargetPower := byManualyTargetPowerUV1_3;
	
fbAlfen3(
	bEnable:= , 
	bPowerDataInvers:= , 
	byElectricFuseLine:= , 
	byUnitID_Socket1:= 1, 
	byUnitID_Socket2:= , 
	byNumberOfSockets:= 1, 
	byNumberOfConnectionWire:= 1, 
	diNrOfEMS_IN:= prgEMS.fbEMS.diNrOfEMS_OUT, 
	diNrOfEM_IN_CS:= , 
	sIPAdress:= '192.168.1.164',  
	stSetupECS:= , 
	stDataECS=> , 
	diNrOfECS_OUT=> );

bSManualyOn_UV1_3 := fbAlfen3.stDataECS.bSManualyOn;
	bySManualyTargetPowerUV1_3 := fbAlfen3.stDataECS.bySManualyTargetPower;
		byErrorWarningUV1_3 := fbAlfen3.stDataECS.byErrorWarning;
			rChargingTimeInMinUV1_3 := fbAlfen3.stDataECS.arrChargingTimeInMin[1];	
				lrPowerUV1_3 := fbAlfen3.stDataECS.lrTotalPower;	
					wStateUV1_3 := fbAlfen3.stDataECS.arrSocketStateECS[1];
						lrEnergySessionUV1_3 := fbAlfen3.stDataECS.arrSocketEnergySession[1];
							lrTotalEnergyUV1_3 := fbAlfen3.stDataECS.lrTotalCounterEnergy_Consumption;	
	
(*---------------------------------------------CS4-----------------------------------------------------------*)	
	
//Manual Power
fbAlfen4.stSetupECS.bManualyOn := bManualyOnUV1_4;
	fbAlfen4.stSetupECS.byManualyTargetPower := byManualyTargetPowerUV1_4;
	
fbAlfen4(
	bEnable:= , 
	bPowerDataInvers:= , 
	byElectricFuseLine:= , 
	byUnitID_Socket1:= 1, 
	byUnitID_Socket2:= , 
	byNumberOfSockets:= 1, 
	byNumberOfConnectionWire:= 1, 
	diNrOfEMS_IN:= prgEMS.fbEMS.diNrOfEMS_OUT, 
	diNrOfEM_IN_CS:= , 
	sIPAdress:= '192.168.1.188',  
	stSetupECS:= , 
	stDataECS=> , 
	diNrOfECS_OUT=> );

bSManualyOn_UV1_4 := fbAlfen4.stDataECS.bSManualyOn;
	bySManualyTargetPowerUV1_4 := fbAlfen4.stDataECS.bySManualyTargetPower;	
		byErrorWarningUV1_4 := fbAlfen4.stDataECS.byErrorWarning;
			rChargingTimeInMinUV1_4 := fbAlfen4.stDataECS.arrChargingTimeInMin[1];
				lrPowerUV1_4 := fbAlfen4.stDataECS.lrTotalPower;	
					wStateUV1_4 := fbAlfen4.stDataECS.arrSocketStateECS[1];
						lrEnergySessionUV1_4 := fbAlfen4.stDataECS.arrSocketEnergySession[1];
							lrTotalEnergyUV1_4 := fbAlfen4.stDataECS.lrTotalCounterEnergy_Consumption;
	
(*---------------------------------------------CS5-----------------------------------------------------------*)	
	
//Manual Power
fbAlfen5.stSetupECS.bManualyOn := bManualyOnUV1_5;
	fbAlfen5.stSetupECS.byManualyTargetPower := byManualyTargetPowerUV1_5;
	
fbAlfen5(
	bEnable:= , 
	bPowerDataInvers:= , 
	byElectricFuseLine:= , 
	byUnitID_Socket1:= 1, 
	byUnitID_Socket2:= , 
	byNumberOfSockets:= 1, 
	byNumberOfConnectionWire:= 1, 
	diNrOfEMS_IN:= prgEMS.fbEMS.diNrOfEMS_OUT, 
	diNrOfEM_IN_CS:= , 
	sIPAdress:= '192.168.1.103',  
	stSetupECS:= , 
	stDataECS=> , 
	diNrOfECS_OUT=> );

bSManualyOn_UV1_5 := fbAlfen5.stDataECS.bSManualyOn;
	bySManualyTargetPowerUV1_5 := fbAlfen5.stDataECS.bySManualyTargetPower;
		byErrorWarningUV1_5 := fbAlfen5.stDataECS.byErrorWarning;
			rChargingTimeInMinUV1_5 := fbAlfen5.stDataECS.arrChargingTimeInMin[1];
				lrPowerUV1_5 := fbAlfen5.stDataECS.lrTotalPower;	
					wStateUV1_5 := fbAlfen5.stDataECS.arrSocketStateECS[1];
						lrEnergySessionUV1_5 := fbAlfen5.stDataECS.arrSocketEnergySession[1];
							lrTotalEnergyUV1_5 := fbAlfen5.stDataECS.lrTotalCounterEnergy_Consumption;	
	
(*---------------------------------------------CS6-----------------------------------------------------------*)	
	
//Manual Power
fbAlfen6.stSetupECS.bManualyOn := bManualyOnUV1_6;
	fbAlfen6.stSetupECS.byManualyTargetPower := byManualyTargetPowerUV1_6;
	
fbAlfen6(
	bEnable:= , 
	bPowerDataInvers:= , 
	byElectricFuseLine:= , 
	byUnitID_Socket1:= 1, 
	byUnitID_Socket2:= , 
	byNumberOfSockets:= 1, 
	byNumberOfConnectionWire:= 1, 
	diNrOfEMS_IN:= prgEMS.fbEMS.diNrOfEMS_OUT, 
	diNrOfEM_IN_CS:= , 
	sIPAdress:= '192.168.1.128',  
	stSetupECS:= , 
	stDataECS=> , 
	diNrOfECS_OUT=> );

bSManualyOn_UV1_6 := fbAlfen6.stDataECS.bSManualyOn;
	bySManualyTargetPowerUV1_6 := fbAlfen6.stDataECS.bySManualyTargetPower;	
		byErrorWarningUV1_6 := fbAlfen6.stDataECS.byErrorWarning;
			rChargingTimeInMinUV1_6 := fbAlfen6.stDataECS.arrChargingTimeInMin[1];
				lrPowerUV1_6 := fbAlfen6.stDataECS.lrTotalPower;	
					wStateUV1_6 := fbAlfen6.stDataECS.arrSocketStateECS[1];
						lrEnergySessionUV1_6 := fbAlfen6.stDataECS.arrSocketEnergySession[1];
							lrTotalEnergyUV1_6 := fbAlfen6.stDataECS.lrTotalCounterEnergy_Consumption;
	
(*---------------------------------------------CS7-----------------------------------------------------------*)	
	
//Manual Power
fbAlfen7.stSetupECS.bManualyOn := bManualyOnUV1_7;
	fbAlfen7.stSetupECS.byManualyTargetPower := byManualyTargetPowerUV1_7;
	
fbAlfen7(
	bEnable:= , 
	bPowerDataInvers:= , 
	byElectricFuseLine:= , 
	byUnitID_Socket1:= 1, 
	byUnitID_Socket2:= , 
	byNumberOfSockets:= 1, 
	byNumberOfConnectionWire:= 1, 
	diNrOfEMS_IN:= prgEMS.fbEMS.diNrOfEMS_OUT, 
	diNrOfEM_IN_CS:= , 
	sIPAdress:= '192.168.1.113',  
	stSetupECS:= , 
	stDataECS=> , 
	diNrOfECS_OUT=> );

bSManualyOn_UV1_7 := fbAlfen7.stDataECS.bSManualyOn;
	bySManualyTargetPowerUV1_7 := fbAlfen7.stDataECS.bySManualyTargetPower;	
		byErrorWarningUV1_7 := fbAlfen7.stDataECS.byErrorWarning;
			rChargingTimeInMinUV1_7 := fbAlfen7.stDataECS.arrChargingTimeInMin[1];
				lrPowerUV1_7 := fbAlfen7.stDataECS.lrTotalPower;	
					wStateUV1_7 := fbAlfen7.stDataECS.arrSocketStateECS[1];
						lrEnergySessionUV1_7 := fbAlfen7.stDataECS.arrSocketEnergySession[1];
							lrTotalEnergyUV1_7 := fbAlfen7.stDataECS.lrTotalCounterEnergy_Consumption;
	
(*---------------------------------------------CS8-----------------------------------------------------------*)	
	
//Manual Power
fbAlfen8.stSetupECS.bManualyOn := bManualyOnUV1_8;
	fbAlfen8.stSetupECS.byManualyTargetPower := byManualyTargetPowerUV1_8;
	
fbAlfen8(
	bEnable:= , 
	bPowerDataInvers:= , 
	byElectricFuseLine:= , 
	byUnitID_Socket1:= 1, 
	byUnitID_Socket2:= , 
	byNumberOfSockets:= 1, 
	byNumberOfConnectionWire:= 1, 
	diNrOfEMS_IN:= prgEMS.fbEMS.diNrOfEMS_OUT, 
	diNrOfEM_IN_CS:= , 
	sIPAdress:= '192.168.1.109',  
	stSetupECS:= , 
	stDataECS=> , 
	diNrOfECS_OUT=> );

bSManualyOn_UV1_8 := fbAlfen8.stDataECS.bSManualyOn;
	bySManualyTargetPowerUV1_8 := fbAlfen8.stDataECS.bySManualyTargetPower;	
		byErrorWarningUV1_8 := fbAlfen8.stDataECS.byErrorWarning;
			rChargingTimeInMinUV1_8 := fbAlfen8.stDataECS.arrChargingTimeInMin[1];
				lrPowerUV1_8 := fbAlfen8.stDataECS.lrTotalPower;	
					wStateUV1_8 := fbAlfen8.stDataECS.arrSocketStateECS[1];
						lrEnergySessionUV1_8 := fbAlfen8.stDataECS.arrSocketEnergySession[1];
							lrTotalEnergyUV1_8 := fbAlfen8.stDataECS.lrTotalCounterEnergy_Consumption;
	
(*---------------------------------------------CS9-----------------------------------------------------------*)	
	
//Manual Power
fbAlfen9.stSetupECS.bManualyOn := bManualyOnUV1_9;
	fbAlfen9.stSetupECS.byManualyTargetPower := byManualyTargetPowerUV1_9;
	
fbAlfen9(
	bEnable:= , 
	bPowerDataInvers:= , 
	byElectricFuseLine:= , 
	byUnitID_Socket1:= 1, 
	byUnitID_Socket2:= , 
	byNumberOfSockets:= 1, 
	byNumberOfConnectionWire:= 1, 
	diNrOfEMS_IN:= prgEMS.fbEMS.diNrOfEMS_OUT, 
	diNrOfEM_IN_CS:= , 
	sIPAdress:= '192.168.1.141',  
	stSetupECS:= , 
	stDataECS=> , 
	diNrOfECS_OUT=> );

bSManualyOn_UV1_9 := fbAlfen9.stDataECS.bSManualyOn;
	bySManualyTargetPowerUV1_9 := fbAlfen9.stDataECS.bySManualyTargetPower;
		byErrorWarningUV1_9 := fbAlfen9.stDataECS.byErrorWarning;	
			rChargingTimeInMinUV1_9 := fbAlfen9.stDataECS.arrChargingTimeInMin[1];
				lrPowerUV1_9 := fbAlfen9.stDataECS.lrTotalPower;	
					wStateUV1_9 := fbAlfen9.stDataECS.arrSocketStateECS[1];
						lrEnergySessionUV1_9 := fbAlfen9.stDataECS.arrSocketEnergySession[1];
							lrTotalEnergyUV1_9 := fbAlfen9.stDataECS.lrTotalCounterEnergy_Consumption;
	
(*---------------------------------------------CS10-----------------------------------------------------------*)	
	
//Manual Power
fbAlfen10.stSetupECS.bManualyOn := bManualyOnUV1_10;
	fbAlfen10.stSetupECS.byManualyTargetPower := byManualyTargetPowerUV1_10;
	
fbAlfen10(
	bEnable:= , 
	bPowerDataInvers:= , 
	byElectricFuseLine:= , 
	byUnitID_Socket1:= 1, 
	byUnitID_Socket2:= , 
	byNumberOfSockets:= 1, 
	byNumberOfConnectionWire:= 1, 
	diNrOfEMS_IN:= prgEMS.fbEMS.diNrOfEMS_OUT, 
	diNrOfEM_IN_CS:= , 
	sIPAdress:= '192.168.1.231', 
	stSetupECS:= , 
	stDataECS=> , 
	diNrOfECS_OUT=> );

bSManualyOn_UV1_10 := fbAlfen10.stDataECS.bSManualyOn;
	bySManualyTargetPowerUV1_10 := fbAlfen10.stDataECS.bySManualyTargetPower;
		byErrorWarningUV1_10 := fbAlfen10.stDataECS.byErrorWarning;	
			rChargingTimeInMinUV1_10 := fbAlfen10.stDataECS.arrChargingTimeInMin[1];
				lrPowerUV1_10 := fbAlfen10.stDataECS.lrTotalPower;	
					wStateUV1_10 := fbAlfen10.stDataECS.arrSocketStateECS[1];
						lrEnergySessionUV1_10 := fbAlfen10.stDataECS.arrSocketEnergySession[1];
							lrTotalEnergyUV1_10 := fbAlfen10.stDataECS.lrTotalCounterEnergy_Consumption;

END_PROGRAM

// ---- POUs/prgCS6.TcPOU
PROGRAM prgCS6
VAR
	fbAlfen1					: FB_ECS_Alfen_NG9xx_Platform;						//{#lynus.ag#()}
	fbAlfen2					: FB_ECS_Alfen_NG9xx_Platform;						//{#lynus.ag#()}
	fbAlfen3					: FB_ECS_Alfen_NG9xx_Platform;						//{#lynus.ag#()}
	fbAlfen4					: FB_ECS_Alfen_NG9xx_Platform;						//{#lynus.ag#()}
	fbAlfen5					: FB_ECS_Alfen_NG9xx_Platform;						//{#lynus.ag#()}
	fbAlfen6					: FB_ECS_Alfen_NG9xx_Platform;						//{#lynus.ag#()}
	fbAlfen7					: FB_ECS_Alfen_NG9xx_Platform;						//{#lynus.ag#()}
	fbAlfen8					: FB_ECS_Alfen_NG9xx_Platform;						//{#lynus.ag#()}
	fbAlfen9					: FB_ECS_Alfen_NG9xx_Platform;						//{#lynus.ag#()}
	fbAlfen10					: FB_ECS_Alfen_NG9xx_Platform;						//{#lynus.ag#()}
	
	bSManualyOn_UV1_1			: BOOL;												//{#lynus.ag#()}
	bySManualyTargetPowerUV1_1	: BYTE;												//{#lynus.ag#()}
	byErrorWarningUV1_1			: BYTE;												//{#lynus.ag#()}
	rChargingTimeInMinUV1_1		: REAL;												//{#lynus.ag#()}
	lrPowerUV1_1				: LREAL;											//{#lynus.ag#()}
	wStateUV1_1					: WORD;												//{#lynus.ag#()}
	lrEnergySessionUV1_1		: LREAL;											//{#lynus.ag#()}
	lrTotalEnergyUV1_1			: LREAL;											//{#lynus.ag#()}
	
	bSManualyOn_UV1_2			: BOOL;												//{#lynus.ag#()}
	bySManualyTargetPowerUV1_2	: BYTE;												//{#lynus.ag#()}
	byErrorWarningUV1_2			: BYTE;												//{#lynus.ag#()}
	rChargingTimeInMinUV1_2		: REAL;												//{#lynus.ag#()}
	lrPowerUV1_2				: LREAL;											//{#lynus.ag#()}
	wStateUV1_2					: WORD;												//{#lynus.ag#()}
	lrEnergySessionUV1_2		: LREAL;											//{#lynus.ag#()}
	lrTotalEnergyUV1_2			: LREAL;											//{#lynus.ag#()}
	
	bSManualyOn_UV1_3			: BOOL;												//{#lynus.ag#()}
	bySManualyTargetPowerUV1_3	: BYTE;												//{#lynus.ag#()}
	byErrorWarningUV1_3			: BYTE;												//{#lynus.ag#()}
	rChargingTimeInMinUV1_3		: REAL;												//{#lynus.ag#()}
	lrPowerUV1_3				: LREAL;											//{#lynus.ag#()}
	wStateUV1_3					: WORD;												//{#lynus.ag#()}
	lrEnergySessionUV1_3		: LREAL;											//{#lynus.ag#()}
	lrTotalEnergyUV1_3			: LREAL;											//{#lynus.ag#()}
	
	bSManualyOn_UV1_4			: BOOL;												//{#lynus.ag#()}
	bySManualyTargetPowerUV1_4	: BYTE;												//{#lynus.ag#()}
	byErrorWarningUV1_4			: BYTE;												//{#lynus.ag#()}
	rChargingTimeInMinUV1_4		: REAL;												//{#lynus.ag#()}
	lrPowerUV1_4				: LREAL;											//{#lynus.ag#()}
	wStateUV1_4					: WORD;												//{#lynus.ag#()}
	lrEnergySessionUV1_4		: LREAL;											//{#lynus.ag#()}
	lrTotalEnergyUV1_4			: LREAL;											//{#lynus.ag#()}
	
	bSManualyOn_UV1_5			: BOOL;												//{#lynus.ag#()}
	bySManualyTargetPowerUV1_5	: BYTE;												//{#lynus.ag#()}
	byErrorWarningUV1_5			: BYTE;												//{#lynus.ag#()}
	rChargingTimeInMinUV1_5		: REAL;												//{#lynus.ag#()}
	lrPowerUV1_5				: LREAL;											//{#lynus.ag#()}
	wStateUV1_5					: WORD;												//{#lynus.ag#()}
	lrEnergySessionUV1_5		: LREAL;											//{#lynus.ag#()}
	lrTotalEnergyUV1_5			: LREAL;											//{#lynus.ag#()}
	
	bSManualyOn_UV1_6			: BOOL;												//{#lynus.ag#()}
	bySManualyTargetPowerUV1_6	: BYTE;												//{#lynus.ag#()}
	byErrorWarningUV1_6			: BYTE;												//{#lynus.ag#()}
	rChargingTimeInMinUV1_6		: REAL;												//{#lynus.ag#()}
	lrPowerUV1_6				: LREAL;											//{#lynus.ag#()}
	wStateUV1_6					: WORD;												//{#lynus.ag#()}
	lrEnergySessionUV1_6		: LREAL;											//{#lynus.ag#()}
	lrTotalEnergyUV1_6			: LREAL;											//{#lynus.ag#()}
	
	bSManualyOn_UV1_7			: BOOL;												//{#lynus.ag#()}
	bySManualyTargetPowerUV1_7	: BYTE;												//{#lynus.ag#()}
	byErrorWarningUV1_7			: BYTE;												//{#lynus.ag#()}
	rChargingTimeInMinUV1_7		: REAL;												//{#lynus.ag#()}
	lrPowerUV1_7				: LREAL;											//{#lynus.ag#()}
	wStateUV1_7					: WORD;												//{#lynus.ag#()}
	lrEnergySessionUV1_7		: LREAL;											//{#lynus.ag#()}
	lrTotalEnergyUV1_7			: LREAL;											//{#lynus.ag#()}
	
	bSManualyOn_UV1_8			: BOOL;												//{#lynus.ag#()}
	bySManualyTargetPowerUV1_8	: BYTE;												//{#lynus.ag#()}
	byErrorWarningUV1_8			: BYTE;												//{#lynus.ag#()}
	rChargingTimeInMinUV1_8		: REAL;												//{#lynus.ag#()}
	lrPowerUV1_8				: LREAL;											//{#lynus.ag#()}
	wStateUV1_8					: WORD;												//{#lynus.ag#()}
	lrEnergySessionUV1_8		: LREAL;											//{#lynus.ag#()}
	lrTotalEnergyUV1_8			: LREAL;											//{#lynus.ag#()}
	
	bSManualyOn_UV1_9			: BOOL;												//{#lynus.ag#()}
	bySManualyTargetPowerUV1_9	: BYTE;												//{#lynus.ag#()}
	byErrorWarningUV1_9			: BYTE;												//{#lynus.ag#()}
	rChargingTimeInMinUV1_9		: REAL;												//{#lynus.ag#()}
	lrPowerUV1_9				: LREAL;											//{#lynus.ag#()}
	wStateUV1_9					: WORD;												//{#lynus.ag#()}
	lrEnergySessionUV1_9		: LREAL;											//{#lynus.ag#()}
	lrTotalEnergyUV1_9			: LREAL;											//{#lynus.ag#()}
	
	bSManualyOn_UV1_10			: BOOL;												//{#lynus.ag#()}
	bySManualyTargetPowerUV1_10	: BYTE;												//{#lynus.ag#()}
	byErrorWarningUV1_10		: BYTE;												//{#lynus.ag#()}
	rChargingTimeInMinUV1_10	: REAL;												//{#lynus.ag#()}
	lrPowerUV1_10				: LREAL;											//{#lynus.ag#()}
	wStateUV1_10				: WORD;												//{#lynus.ag#()}
	lrEnergySessionUV1_10		: LREAL;											//{#lynus.ag#()}
	lrTotalEnergyUV1_10			: LREAL;											//{#lynus.ag#()}
END_VAR
VAR PERSISTENT
	bManualyOnUV1_1				: BOOL;												//{#lynus.ag#()}
	byManualyTargetPowerUV1_1	: BYTE;												//{#lynus.ag#()}
	
	bManualyOnUV1_2				: BOOL;												//{#lynus.ag#()}
	byManualyTargetPowerUV1_2	: BYTE;												//{#lynus.ag#()}
	
	bManualyOnUV1_3				: BOOL;												//{#lynus.ag#()}
	byManualyTargetPowerUV1_3	: BYTE;												//{#lynus.ag#()}
	
	bManualyOnUV1_4				: BOOL;												//{#lynus.ag#()}
	byManualyTargetPowerUV1_4	: BYTE;												//{#lynus.ag#()}
	
	bManualyOnUV1_5				: BOOL;												//{#lynus.ag#()}
	byManualyTargetPowerUV1_5	: BYTE;												//{#lynus.ag#()}
	
	bManualyOnUV1_6				: BOOL;												//{#lynus.ag#()}
	byManualyTargetPowerUV1_6	: BYTE;												//{#lynus.ag#()}
	
	bManualyOnUV1_7				: BOOL;												//{#lynus.ag#()}
	byManualyTargetPowerUV1_7	: BYTE;												//{#lynus.ag#()}
	
	bManualyOnUV1_8				: BOOL;												//{#lynus.ag#()}
	byManualyTargetPowerUV1_8	: BYTE;												//{#lynus.ag#()}
	
	bManualyOnUV1_9				: BOOL;												//{#lynus.ag#()}
	byManualyTargetPowerUV1_9	: BYTE;												//{#lynus.ag#()}
	
	bManualyOnUV1_10			: BOOL;												//{#lynus.ag#()}
	byManualyTargetPowerUV1_10	: BYTE;												//{#lynus.ag#()}
END_VAR

(*---------------------------------------------CS1-----------------------------------------------------------*)

//Manual Power
fbAlfen1.stSetupECS.bManualyOn := bManualyOnUV1_1;
	fbAlfen1.stSetupECS.byManualyTargetPower := byManualyTargetPowerUV1_1;

fbAlfen1(
	bEnable:= , 
	bPowerDataInvers:= , 
	byElectricFuseLine:= , 
	byUnitID_Socket1:= 1, 
	byUnitID_Socket2:= , 
	byNumberOfSockets:= 1, 
	byNumberOfConnectionWire:= 1, 
	diNrOfEMS_IN:= prgEMS.fbEMS.diNrOfEMS_OUT, 
	diNrOfEM_IN_CS:= , 
	sIPAdress:= '192.168.1.143', 
	stSetupECS:= , 
	stDataECS=> , 
	diNrOfECS_OUT=> );

bSManualyOn_UV1_1 := fbAlfen1.stDataECS.bSManualyOn;
	bySManualyTargetPowerUV1_1 := fbAlfen1.stDataECS.bySManualyTargetPower;
		byErrorWarningUV1_1 := fbAlfen1.stDataECS.byErrorWarning;	
			rChargingTimeInMinUV1_1 := fbAlfen1.stDataECS.arrChargingTimeInMin[1];
				lrPowerUV1_1 := fbAlfen1.stDataECS.lrTotalPower;	
					wStateUV1_1 := fbAlfen1.stDataECS.arrSocketStateECS[1];
						lrEnergySessionUV1_1 := fbAlfen1.stDataECS.arrSocketEnergySession[1];
							lrTotalEnergyUV1_1 := fbAlfen1.stDataECS.lrTotalCounterEnergy_Consumption;	
	
(*---------------------------------------------CS2-----------------------------------------------------------*)
	
//Manual Power
fbAlfen2.stSetupECS.bManualyOn := bManualyOnUV1_2;
	fbAlfen2.stSetupECS.byManualyTargetPower := byManualyTargetPowerUV1_2;
	
fbAlfen2(
	bEnable:= , 
	bPowerDataInvers:= , 
	byElectricFuseLine:= , 
	byUnitID_Socket1:= 1, 
	byUnitID_Socket2:= , 
	byNumberOfSockets:= 1, 
	byNumberOfConnectionWire:= 1, 
	diNrOfEMS_IN:= prgEMS.fbEMS.diNrOfEMS_OUT, 
	diNrOfEM_IN_CS:= , 
	sIPAdress:= '192.168.1.162', 
	stSetupECS:= , 
	stDataECS=> , 
	diNrOfECS_OUT=> );

bSManualyOn_UV1_2 := fbAlfen2.stDataECS.bSManualyOn;
	bySManualyTargetPowerUV1_2 := fbAlfen2.stDataECS.bySManualyTargetPower;	
		byErrorWarningUV1_2 := fbAlfen2.stDataECS.byErrorWarning;
			rChargingTimeInMinUV1_2 := fbAlfen2.stDataECS.arrChargingTimeInMin[1];;
				lrPowerUV1_2 := fbAlfen2.stDataECS.lrTotalPower;	
					wStateUV1_2 := fbAlfen2.stDataECS.arrSocketStateECS[1];
						lrEnergySessionUV1_2 := fbAlfen2.stDataECS.arrSocketEnergySession[1];
							lrTotalEnergyUV1_2 := fbAlfen2.stDataECS.lrTotalCounterEnergy_Consumption;
	
(*---------------------------------------------CS3-----------------------------------------------------------*)	
	
//Manual Power
fbAlfen3.stSetupECS.bManualyOn := bManualyOnUV1_3;
	fbAlfen3.stSetupECS.byManualyTargetPower := byManualyTargetPowerUV1_3;
	
fbAlfen3(
	bEnable:= , 
	bPowerDataInvers:= , 
	byElectricFuseLine:= , 
	byUnitID_Socket1:= 1, 
	byUnitID_Socket2:= , 
	byNumberOfSockets:= 1, 
	byNumberOfConnectionWire:= 1, 
	diNrOfEMS_IN:= prgEMS.fbEMS.diNrOfEMS_OUT, 
	diNrOfEM_IN_CS:= , 
	sIPAdress:= '192.168.1.187',  
	stSetupECS:= , 
	stDataECS=> , 
	diNrOfECS_OUT=> );

bSManualyOn_UV1_3 := fbAlfen3.stDataECS.bSManualyOn;
	bySManualyTargetPowerUV1_3 := fbAlfen3.stDataECS.bySManualyTargetPower;
		byErrorWarningUV1_3 := fbAlfen3.stDataECS.byErrorWarning;
			rChargingTimeInMinUV1_3 := fbAlfen3.stDataECS.arrChargingTimeInMin[1];	
				lrPowerUV1_3 := fbAlfen3.stDataECS.lrTotalPower;	
					wStateUV1_3 := fbAlfen3.stDataECS.arrSocketStateECS[1];
						lrEnergySessionUV1_3 := fbAlfen3.stDataECS.arrSocketEnergySession[1];
							lrTotalEnergyUV1_3 := fbAlfen3.stDataECS.lrTotalCounterEnergy_Consumption;	
	
(*---------------------------------------------CS4-----------------------------------------------------------*)	
	
//Manual Power
fbAlfen4.stSetupECS.bManualyOn := bManualyOnUV1_4;
	fbAlfen4.stSetupECS.byManualyTargetPower := byManualyTargetPowerUV1_4;
	
fbAlfen4(
	bEnable:= , 
	bPowerDataInvers:= , 
	byElectricFuseLine:= , 
	byUnitID_Socket1:= 1, 
	byUnitID_Socket2:= , 
	byNumberOfSockets:= 1, 
	byNumberOfConnectionWire:= 1, 
	diNrOfEMS_IN:= prgEMS.fbEMS.diNrOfEMS_OUT, 
	diNrOfEM_IN_CS:= , 
	sIPAdress:= '192.168.1.108',  
	stSetupECS:= , 
	stDataECS=> , 
	diNrOfECS_OUT=> );

bSManualyOn_UV1_4 := fbAlfen4.stDataECS.bSManualyOn;
	bySManualyTargetPowerUV1_4 := fbAlfen4.stDataECS.bySManualyTargetPower;	
		byErrorWarningUV1_4 := fbAlfen4.stDataECS.byErrorWarning;
			rChargingTimeInMinUV1_4 := fbAlfen4.stDataECS.arrChargingTimeInMin[1];
				lrPowerUV1_4 := fbAlfen4.stDataECS.lrTotalPower;	
					wStateUV1_4 := fbAlfen4.stDataECS.arrSocketStateECS[1];
						lrEnergySessionUV1_4 := fbAlfen4.stDataECS.arrSocketEnergySession[1];
							lrTotalEnergyUV1_4 := fbAlfen4.stDataECS.lrTotalCounterEnergy_Consumption;
	
(*---------------------------------------------CS5-----------------------------------------------------------*)	
	
//Manual Power
fbAlfen5.stSetupECS.bManualyOn := bManualyOnUV1_5;
	fbAlfen5.stSetupECS.byManualyTargetPower := byManualyTargetPowerUV1_5;
	
fbAlfen5(
	bEnable:= , 
	bPowerDataInvers:= , 
	byElectricFuseLine:= , 
	byUnitID_Socket1:= 1, 
	byUnitID_Socket2:= , 
	byNumberOfSockets:= 1, 
	byNumberOfConnectionWire:= 1, 
	diNrOfEMS_IN:= prgEMS.fbEMS.diNrOfEMS_OUT, 
	diNrOfEM_IN_CS:= , 
	sIPAdress:= '192.168.1.150',  
	stSetupECS:= , 
	stDataECS=> , 
	diNrOfECS_OUT=> );

bSManualyOn_UV1_5 := fbAlfen5.stDataECS.bSManualyOn;
	bySManualyTargetPowerUV1_5 := fbAlfen5.stDataECS.bySManualyTargetPower;
		byErrorWarningUV1_5 := fbAlfen5.stDataECS.byErrorWarning;
			rChargingTimeInMinUV1_5 := fbAlfen5.stDataECS.arrChargingTimeInMin[1];
				lrPowerUV1_5 := fbAlfen5.stDataECS.lrTotalPower;	
					wStateUV1_5 := fbAlfen5.stDataECS.arrSocketStateECS[1];
						lrEnergySessionUV1_5 := fbAlfen5.stDataECS.arrSocketEnergySession[1];
							lrTotalEnergyUV1_5 := fbAlfen5.stDataECS.lrTotalCounterEnergy_Consumption;		
	
(*---------------------------------------------CS6-----------------------------------------------------------*)	
	
//Manual Power
fbAlfen6.stSetupECS.bManualyOn := bManualyOnUV1_6;
	fbAlfen6.stSetupECS.byManualyTargetPower := byManualyTargetPowerUV1_6;
	
fbAlfen6(
	bEnable:= , 
	bPowerDataInvers:= , 
	byElectricFuseLine:= , 
	byUnitID_Socket1:= 1, 
	byUnitID_Socket2:= , 
	byNumberOfSockets:= 1, 
	byNumberOfConnectionWire:= 1, 
	diNrOfEMS_IN:= prgEMS.fbEMS.diNrOfEMS_OUT, 
	diNrOfEM_IN_CS:= , 
	sIPAdress:= '192.168.1.114',  
	stSetupECS:= , 
	stDataECS=> , 
	diNrOfECS_OUT=> );

